C05487=1178.602,249.127,-64.757,-177.311,7.252,148.580
C05488=1178.597,249.375,-64.784,-177.309,7.254,148.579
C05489=1178.592,249.624,-64.811,-177.306,7.257,148.579
C05490=1178.588,249.872,-64.838,-177.303,7.259,148.579
C05491=1178.584,250.121,-64.865,-177.301,7.262,148.579
C05492=1178.580,250.370,-64.892,-177.299,7.264,148.579
C05493=1178.575,250.618,-64.919,-177.295,7.267,148.579
C05494=1178.571,250.866,-64.946,-177.293,7.270,148.579
C05495=1178.566,251.115,-64.973,-177.290,7.272,148.578
C05496=1178.562,251.363,-65.000,-177.288,7.275,148.578
C05497=1178.557,251.612,-65.027,-177.285,7.276,148.578
C05498=1178.553,251.860,-65.054,-177.282,7.279,148.578
C05499=1178.549,252.109,-65.081,-177.280,7.282,148.578
C05500=1178.545,252.358,-65.108,-177.277,7.285,148.578
C05501=1178.540,252.606,-65.135,-177.274,7.287,148.578
C05502=1178.536,252.854,-65.163,-177.272,7.289,148.577
C05503=1178.531,253.103,-65.190,-177.269,7.292,148.577
C05504=1178.526,253.351,-65.217,-177.267,7.295,148.577
C05505=1178.522,253.600,-65.244,-177.264,7.297,148.577
C05506=1178.518,253.849,-65.271,-177.261,7.300,148.577
C05507=1178.514,254.097,-65.298,-177.259,7.302,148.577
C05508=1178.509,254.345,-65.326,-177.256,7.305,148.577
C05509=1178.505,254.593,-65.353,-177.253,7.308,148.577
C05510=1178.500,254.842,-65.380,-177.251,7.310,148.576
C05511=1178.496,255.091,-65.407,-177.248,7.313,148.576
C05512=1178.492,255.339,-65.435,-177.245,7.316,148.576
C05513=1178.487,255.588,-65.462,-177.243,7.318,148.576
C05514=1178.482,255.836,-65.489,-177.240,7.321,148.576
C05515=1178.478,256.085,-65.517,-177.238,7.323,148.576
C05516=1178.474,256.333,-65.544,-177.235,7.326,148.576
C05517=1178.469,256.582,-65.571,-177.232,7.329,148.576
C05518=1178.464,256.830,-65.598,-177.230,7.331,148.575
C05519=1178.461,257.079,-65.627,-177.227,7.334,148.575
C05520=1178.456,257.327,-65.654,-177.224,7.337,148.575
C05521=1178.451,257.576,-65.681,-177.222,7.339,148.575
C05522=1178.447,257.824,-65.708,-177.219,7.342,148.575
C05523=1178.443,258.073,-65.736,-177.216,7.344,148.575
C05524=1178.438,258.321,-65.763,-177.214,7.347,148.575
C05525=1178.434,258.569,-65.791,-177.211,7.350,148.575
C05526=1178.429,258.818,-65.818,-177.209,7.352,148.575
C05527=1178.426,259.066,-65.846,-177.206,7.355,148.575
C05528=1178.421,259.315,-65.873,-177.204,7.358,148.575
C05529=1178.417,259.563,-65.901,-177.201,7.359,148.574
C05530=1178.413,259.812,-65.928,-177.198,7.362,148.574
C05531=1178.408,260.060,-65.956,-177.195,7.365,148.574
C05532=1178.404,260.308,-65.983,-177.193,7.368,148.574
C05533=1178.400,260.557,-66.011,-177.191,7.371,148.574
C05534=1178.394,260.805,-66.039,-177.188,7.373,148.574
C05535=1178.390,261.053,-66.067,-177.185,7.375,148.574
C05536=1178.386,261.303,-66.094,-177.182,7.378,148.574
C05537=1178.382,261.550,-66.122,-177.180,7.381,148.574
C05538=1178.377,261.799,-66.149,-177.177,7.383,148.573
C05539=1178.372,262.072,-66.180,-177.175,7.386,148.573
C05540=1178.367,262.345,-66.210,-177.172,7.389,148.573
C05541=1178.362,262.618,-66.241,-177.169,7.392,148.573
C05542=1178.358,262.891,-66.272,-177.165,7.396,148.573
C05543=1178.353,263.139,-66.299,-177.163,7.398,148.573
C05544=1178.349,263.387,-66.327,-177.161,7.401,148.573
C05545=1178.345,263.636,-66.354,-177.157,7.404,148.573
C05546=1178.341,263.884,-66.382,-177.155,7.406,148.573
C05547=1178.336,264.133,-66.411,-177.152,7.409,148.573
C05548=1178.332,264.381,-66.439,-177.150,7.412,148.573
C05549=1178.327,264.630,-66.466,-177.148,7.414,148.572
C05550=1178.323,264.878,-66.494,-177.145,7.417,148.572
C05551=1178.318,265.126,-66.522,-177.142,7.420,148.572
C05552=1178.315,265.375,-66.550,-177.140,7.422,148.572
C05553=1178.310,265.623,-66.577,-177.137,7.425,148.572
C05554=1178.306,265.871,-66.605,-177.134,7.428,148.572
C05555=1178.301,266.120,-66.634,-177.132,7.430,148.572
C05556=1178.297,266.368,-66.662,-177.129,7.433,148.572
C05557=1178.293,266.617,-66.690,-177.126,7.436,148.572
C05558=1178.288,266.865,-66.717,-177.124,7.439,148.572
C05559=1178.284,267.114,-66.746,-177.121,7.441,148.572
C05560=1178.279,267.362,-66.773,-177.119,7.444,148.572
C05561=1178.274,267.610,-66.802,-177.116,7.447,148.572
C05562=1178.271,267.859,-66.830,-177.114,7.449,148.571
C05563=1178.266,268.107,-66.858,-177.111,7.452,148.571
C05564=1178.262,268.355,-66.886,-177.108,7.455,148.571
C05565=1178.257,268.603,-66.914,-177.105,7.458,148.571
C05566=1178.253,268.853,-66.942,-177.103,7.460,148.571
C05567=1178.248,269.101,-66.970,-177.100,7.463,148.571
C05568=1178.245,269.349,-66.998,-177.097,7.466,148.571
C05569=1178.239,269.597,-67.026,-177.095,7.468,148.571
C05570=1178.236,269.846,-67.055,-177.093,7.471,148.571
C05571=1178.231,270.094,-67.083,-177.090,7.474,148.571
C05572=1178.227,270.343,-67.111,-177.087,7.477,148.571
C05573=1178.223,270.591,-67.139,-177.085,7.479,148.571
C05574=1178.218,270.840,-67.168,-177.082,7.482,148.571
C05575=1178.214,271.087,-67.195,-177.079,7.485,148.570
C05576=1178.209,271.336,-67.225,-177.077,7.487,148.570
C05577=1178.206,271.584,-67.253,-177.075,7.490,148.570
C05578=1178.201,271.832,-67.281,-177.072,7.493,148.570
C05579=1178.197,272.081,-67.309,-177.069,7.496,148.570
C05580=1178.192,272.329,-67.338,-177.066,7.498,148.570
C05581=1178.188,272.578,-67.366,-177.064,7.501,148.570
C05582=1178.183,272.826,-67.394,-177.061,7.504,148.570
C05583=1178.179,273.075,-67.423,-177.058,7.507,148.570
C05584=1178.174,273.322,-67.452,-177.056,7.509,148.570
C05585=1178.171,273.571,-67.480,-177.053,7.512,148.570
C05586=1178.166,273.820,-67.508,-177.051,7.515,148.570
C05587=1178.161,274.068,-67.537,-177.048,7.518,148.570
C05588=1178.157,274.316,-67.565,-177.046,7.520,148.570
C05589=1178.153,274.564,-67.594,-177.043,7.523,148.569
C05590=1178.149,274.813,-67.622,-177.040,7.526,148.569
C05591=1178.144,275.061,-67.651,-177.037,7.529,148.569
C05592=1178.140,275.309,-67.679,-177.035,7.531,148.569
C05593=1178.136,275.558,-67.708,-177.033,7.534,148.569
C05594=1178.131,275.806,-67.737,-177.030,7.537,148.569
C05595=1178.127,276.054,-67.765,-177.027,7.540,148.569
C05596=1178.123,276.303,-67.794,-177.025,7.542,148.569
C05597=1178.118,276.550,-67.822,-177.022,7.545,148.569
C05598=1178.114,276.799,-67.851,-177.019,7.548,148.569
C05599=1178.110,277.048,-67.880,-177.017,7.551,148.569
C05600=1178.105,277.295,-67.908,-177.015,7.553,148.569
C05601=1178.101,277.544,-67.937,-177.012,7.556,148.569
C05602=1178.097,277.793,-67.966,-177.009,7.559,148.569
C05603=1178.093,278.041,-67.994,-177.006,7.562,148.569
C05604=1178.088,278.289,-68.023,-177.004,7.565,148.569
C05605=1178.084,278.538,-68.052,-177.001,7.567,148.569
C05606=1178.080,278.786,-68.082,-176.999,7.570,148.569
C05607=1178.075,279.034,-68.109,-176.996,7.573,148.569
C05608=1178.071,279.283,-68.138,-176.993,7.576,148.569
C05609=1178.067,279.531,-68.167,-176.991,7.578,148.568
C05610=1178.062,279.779,-68.195,-176.988,7.581,148.568
C05611=1178.058,280.027,-68.225,-176.986,7.584,148.568
C05612=1178.054,280.275,-68.254,-176.983,7.587,148.568
C05613=1178.049,280.524,-68.283,-176.980,7.590,148.568
C05614=1178.045,280.772,-68.311,-176.978,7.592,148.568
C05615=1178.041,281.020,-68.340,-176.975,7.595,148.568
C05616=1178.037,281.269,-68.370,-176.973,7.598,148.568
C05617=1178.032,281.518,-68.398,-176.970,7.602,148.568
C05618=1178.027,281.765,-68.427,-176.968,7.604,148.568
C05619=1178.023,282.013,-68.457,-176.965,7.607,148.568
C05620=1178.019,282.262,-68.485,-176.963,7.610,148.568
C05621=1178.015,282.510,-68.514,-176.960,7.613,148.568
C05622=1178.010,282.758,-68.543,-176.957,7.616,148.568
C05623=1178.006,283.007,-68.572,-176.955,7.618,148.568
C05624=1178.002,283.255,-68.602,-176.952,7.621,148.568
C05625=1177.998,283.503,-68.631,-176.950,7.624,148.568
C05626=1177.993,283.751,-68.660,-176.947,7.627,148.568
C05627=1177.988,284.000,-68.689,-176.944,7.630,148.568
C05628=1177.985,284.248,-68.718,-176.942,7.632,148.568
C05629=1177.980,284.497,-68.747,-176.939,7.635,148.568
C05630=1177.976,284.745,-68.776,-176.936,7.638,148.568
C05631=1177.971,284.992,-68.805,-176.934,7.641,148.568
C05632=1177.967,285.241,-68.835,-176.931,7.644,148.568
C05633=1177.963,285.489,-68.864,-176.929,7.647,148.568
C05634=1177.959,285.738,-68.893,-176.927,7.649,148.568
C05635=1177.954,285.986,-68.922,-176.924,7.652,148.568
C05636=1177.950,286.234,-68.952,-176.921,7.655,148.568
C05637=1177.945,286.482,-68.981,-176.918,7.658,148.568
C05638=1177.941,286.730,-69.010,-176.916,7.661,148.568
C05639=1177.937,286.978,-69.040,-176.913,7.664,148.568
C05640=1177.933,287.227,-69.069,-176.911,7.667,148.568
C05641=1177.928,287.476,-69.098,-176.908,7.670,148.567
C05642=1177.924,287.724,-69.127,-176.905,7.673,148.567
C05643=1177.920,287.998,-69.160,-176.903,7.675,148.567
C05644=1177.915,288.273,-69.192,-176.900,7.679,148.568
C05645=1177.910,288.548,-69.226,-176.897,7.683,148.568
C05646=1177.905,288.822,-69.257,-176.894,7.686,148.568
C05647=1177.901,289.070,-69.287,-176.892,7.689,148.568
C05648=1177.897,289.319,-69.316,-176.889,7.692,148.568
C05649=1177.892,289.567,-69.346,-176.887,7.694,148.567
C05650=1177.888,289.815,-69.376,-176.884,7.697,148.567
C05651=1177.884,290.064,-69.405,-176.881,7.700,148.567
C05652=1177.880,290.312,-69.435,-176.878,7.703,148.567
C05653=1177.875,290.560,-69.464,-176.876,7.706,148.567
C05654=1177.871,290.809,-69.493,-176.873,7.709,148.567
C05655=1177.867,291.057,-69.523,-176.871,7.711,148.567
C05656=1177.863,291.304,-69.553,-176.869,7.714,148.567
C05657=1177.858,291.552,-69.582,-176.866,7.717,148.567
C05658=1177.853,291.801,-69.612,-176.863,7.720,148.567
C05659=1177.849,292.049,-69.642,-176.860,7.723,148.567
C05660=1177.845,292.297,-69.671,-176.858,7.726,148.567
C05661=1177.841,292.545,-69.701,-176.855,7.729,148.567
C05662=1177.837,292.794,-69.730,-176.853,7.732,148.567
C05663=1177.833,293.041,-69.760,-176.850,7.734,148.567
C05664=1177.828,293.290,-69.790,-176.848,7.737,148.567
C05665=1177.824,293.538,-69.820,-176.845,7.740,148.567
C05666=1177.820,293.786,-69.849,-176.842,7.743,148.567
C05667=1177.816,294.034,-69.879,-176.840,7.747,148.567
C05668=1177.811,294.283,-69.909,-176.837,7.750,148.567
C05669=1177.807,294.531,-69.939,-176.835,7.752,148.567
C05670=1177.802,294.779,-69.968,-176.832,7.755,148.567
C05671=1177.798,295.027,-69.998,-176.830,7.758,148.567
C05672=1177.794,295.275,-70.029,-176.827,7.761,148.567
C05673=1177.789,295.524,-70.058,-176.825,7.764,148.567
C05674=1177.785,295.771,-70.088,-176.822,7.767,148.567
C05675=1177.782,296.020,-70.118,-176.819,7.770,148.567
C05676=1177.777,296.269,-70.148,-176.816,7.773,148.567
C05677=1177.773,296.517,-70.178,-176.814,7.775,148.567
C05678=1177.769,296.765,-70.208,-176.812,7.779,148.567
C05679=1177.764,297.013,-70.238,-176.809,7.782,148.567
C05680=1177.760,297.261,-70.268,-176.807,7.785,148.567
C05681=1177.756,297.509,-70.297,-176.804,7.788,148.567
C05682=1177.751,297.757,-70.328,-176.801,7.791,148.567
C05683=1177.747,298.006,-70.358,-176.799,7.794,148.568
C05684=1177.743,298.253,-70.388,-176.796,7.797,148.568
C05685=1177.738,298.502,-70.418,-176.794,7.799,148.567
C05686=1177.734,298.749,-70.448,-176.791,7.802,148.567
C05687=1177.730,298.998,-70.478,-176.789,7.805,148.568
C05688=1177.726,299.246,-70.508,-176.786,7.808,148.568
C05689=1177.722,299.495,-70.538,-176.784,7.811,148.568
C05690=1177.718,299.743,-70.569,-176.781,7.814,148.568
C05691=1177.714,299.990,-70.599,-176.778,7.817,148.568
C05692=1177.709,300.239,-70.629,-176.776,7.821,148.568
C05693=1177.705,300.486,-70.659,-176.773,7.824,148.568
C05694=1177.700,300.735,-70.689,-176.771,7.826,148.568
C05695=1177.697,300.983,-70.720,-176.768,7.829,148.568
C05696=1177.692,301.231,-70.750,-176.766,7.832,148.568
C05697=1177.688,301.480,-70.780,-176.763,7.835,148.568
C05698=1177.684,301.727,-70.810,-176.760,7.838,148.568
C05699=1177.679,301.976,-70.840,-176.758,7.841,148.568
C05700=1177.675,302.223,-70.870,-176.755,7.844,148.568
C05701=1177.671,302.471,-70.901,-176.753,7.847,148.568
C05702=1177.667,302.720,-70.932,-176.750,7.850,148.568
C05703=1177.662,302.968,-70.962,-176.747,7.853,148.568
C05704=1177.658,303.216,-70.992,-176.746,7.856,148.568
C05705=1177.654,303.464,-71.023,-176.743,7.859,148.568
C05706=1177.649,303.712,-71.053,-176.740,7.862,148.568
C05707=1177.646,303.961,-71.083,-176.738,7.865,148.568
C05708=1177.641,304.209,-71.114,-176.735,7.868,148.568
C05709=1177.636,304.457,-71.145,-176.732,7.871,148.568
C05710=1177.633,304.704,-71.175,-176.730,7.874,148.568
C05711=1177.628,304.953,-71.205,-176.727,7.877,148.568
C05712=1177.624,305.201,-71.235,-176.725,7.880,148.568
C05713=1177.620,305.449,-71.266,-176.722,7.883,148.568
C05714=1177.615,305.697,-71.297,-176.720,7.887,148.568
C05715=1177.611,305.945,-71.327,-176.717,7.890,148.568
C05716=1177.607,306.194,-71.358,-176.715,7.892,148.568
C05717=1177.603,306.442,-71.389,-176.712,7.895,148.568
C05718=1177.599,306.689,-71.419,-176.710,7.898,148.569
C05719=1177.594,306.937,-71.450,-176.707,7.901,148.568
C05720=1177.590,307.186,-71.480,-176.704,7.904,148.568
C05721=1177.586,307.434,-71.511,-176.702,7.907,148.569
C05722=1177.581,307.682,-71.541,-176.699,7.910,148.569
C05723=1177.577,307.930,-71.572,-176.697,7.913,148.569
C05724=1177.573,308.178,-71.603,-176.694,7.917,148.569
C05725=1177.569,308.426,-71.633,-176.692,7.920,148.569
C05726=1177.564,308.674,-71.664,-176.689,7.923,148.569
C05727=1177.560,308.923,-71.695,-176.687,7.926,148.569
C05728=1177.557,309.170,-71.726,-176.684,7.929,148.569
C05729=1177.552,309.418,-71.757,-176.681,7.932,148.569
C05730=1177.548,309.667,-71.788,-176.679,7.934,148.569
C05731=1177.543,309.914,-71.819,-176.677,7.937,148.569
C05732=1177.540,310.162,-71.849,-176.674,7.940,148.569
C05733=1177.536,310.411,-71.880,-176.672,7.944,148.569
C05734=1177.531,310.659,-71.911,-176.669,7.947,148.569
C05735=1177.526,310.907,-71.942,-176.666,7.950,148.569
C05736=1177.522,311.155,-71.973,-176.664,7.953,148.569
C05737=1177.519,311.402,-72.004,-176.661,7.956,148.569
C05738=1177.514,311.650,-72.034,-176.659,7.959,148.569
C05739=1177.510,311.899,-72.066,-176.656,7.962,148.570
C05740=1177.505,312.147,-72.096,-176.654,7.965,148.570
C05741=1177.501,312.395,-72.127,-176.651,7.968,148.570
C05742=1177.497,312.643,-72.159,-176.649,7.971,148.570
C05743=1177.493,312.891,-72.190,-176.646,7.974,148.570
C05744=1177.489,313.139,-72.220,-176.644,7.978,148.570
C05745=1177.485,313.387,-72.251,-176.641,7.981,148.570
C05746=1177.480,313.635,-72.282,-176.639,7.984,148.570
C05747=1177.475,313.912,-72.317,-176.636,7.987,148.570
C05748=1177.471,314.189,-72.352,-176.633,7.990,148.570
C05749=1177.466,314.465,-72.387,-176.630,7.994,148.570
C05750=1177.462,314.742,-72.421,-176.628,7.997,148.570
C05751=1177.458,314.990,-72.453,-176.625,8.000,148.570
C05752=1177.453,315.238,-72.483,-176.623,8.003,148.570
C05753=1177.449,315.486,-72.515,-176.620,8.006,148.570
C05754=1177.445,315.734,-72.546,-176.617,8.009,148.570
C05755=1177.440,315.982,-72.577,-176.615,8.013,148.571
C05756=1177.437,316.230,-72.609,-176.612,8.016,148.571
C05757=1177.432,316.478,-72.639,-176.610,8.019,148.571
C05758=1177.428,316.726,-72.671,-176.607,8.022,148.571
C05759=1177.424,316.974,-72.702,-176.605,8.025,148.571
C05760=1177.420,317.222,-72.734,-176.602,8.028,148.571
C05761=1177.415,317.470,-72.765,-176.599,8.031,148.571
C05762=1177.412,317.718,-72.796,-176.597,8.035,148.571
C05763=1177.407,317.966,-72.827,-176.594,8.038,148.571
C05764=1177.403,318.214,-72.859,-176.592,8.041,148.571
C05765=1177.399,318.462,-72.890,-176.589,8.044,148.571
C05766=1177.395,318.710,-72.922,-176.587,8.047,148.572
C05767=1177.391,318.958,-72.953,-176.584,8.050,148.572
C05768=1177.387,319.206,-72.984,-176.582,8.053,148.572
C05769=1177.382,319.454,-73.016,-176.579,8.056,148.572
C05770=1177.378,319.703,-73.047,-176.577,8.060,148.572
C05771=1177.373,319.950,-73.079,-176.574,8.063,148.572
C05772=1177.370,320.198,-73.111,-176.572,8.066,148.572
C05773=1177.365,320.446,-73.142,-176.569,8.069,148.572
C05774=1177.361,320.694,-73.173,-176.567,8.072,148.572
C05775=1177.358,320.942,-73.205,-176.564,8.075,148.572
C05776=1177.353,321.190,-73.236,-176.562,8.079,148.573
C05777=1177.349,321.438,-73.268,-176.559,8.082,148.573
C05778=1177.344,321.686,-73.300,-176.557,8.085,148.573
C05779=1177.340,321.934,-73.331,-176.555,8.088,148.573
C05780=1177.336,322.182,-73.363,-176.552,8.091,148.573
C05781=1177.332,322.430,-73.394,-176.550,8.094,148.573
C05782=1177.328,322.678,-73.426,-176.547,8.098,148.573
C05783=1177.324,322.925,-73.458,-176.545,8.101,148.573
C05784=1177.319,323.174,-73.489,-176.542,8.104,148.573
C05785=1177.315,323.422,-73.521,-176.540,8.107,148.573
C05786=1177.311,323.670,-73.553,-176.537,8.110,148.574
C05787=1177.308,323.918,-73.585,-176.535,8.113,148.574
C05788=1177.303,324.165,-73.617,-176.532,8.116,148.574
C05789=1177.299,324.413,-73.649,-176.530,8.119,148.574
C05790=1177.295,324.662,-73.680,-176.527,8.123,148.574
C05791=1177.291,324.909,-73.711,-176.525,8.126,148.574
C05792=1177.286,325.158,-73.744,-176.522,8.129,148.574
C05793=1177.282,325.406,-73.775,-176.520,8.132,148.574
C05794=1177.278,325.653,-73.807,-176.517,8.135,148.574
C05795=1177.274,325.901,-73.839,-176.515,8.139,148.575
C05796=1177.270,326.149,-73.871,-176.512,8.142,148.574
C05797=1177.266,326.397,-73.903,-176.510,8.145,148.575
C05798=1177.261,326.645,-73.935,-176.507,8.148,148.575
C05799=1177.258,326.893,-73.967,-176.505,8.151,148.575
C05800=1177.253,327.140,-73.998,-176.503,8.155,148.575
C05801=1177.249,327.389,-74.031,-176.500,8.158,148.575
C05802=1177.245,327.637,-74.063,-176.498,8.161,148.575
C05803=1177.241,327.884,-74.094,-176.495,8.164,148.575
C05804=1177.236,328.133,-74.127,-176.493,8.167,148.576
C05805=1177.233,328.381,-74.158,-176.491,8.171,148.576
C05806=1177.228,328.628,-74.190,-176.488,8.174,148.576
C05807=1177.224,328.876,-74.222,-176.486,8.177,148.576
C05808=1177.221,329.124,-74.255,-176.483,8.180,148.576
C05809=1177.216,329.372,-74.287,-176.481,8.183,148.576
C05810=1177.212,329.619,-74.319,-176.478,8.186,148.576
C05811=1177.207,329.868,-74.351,-176.476,8.189,148.576
C05812=1177.204,330.116,-74.383,-176.473,8.193,148.577
C05813=1177.199,330.364,-74.416,-176.471,8.196,148.577
C05814=1177.195,330.611,-74.448,-176.468,8.199,148.577
C05815=1177.191,330.859,-74.480,-176.466,8.202,148.577
C05816=1177.187,331.107,-74.512,-176.464,8.206,148.577
C05817=1177.183,331.356,-74.545,-176.461,8.209,148.577
C05818=1177.179,331.602,-74.577,-176.459,8.212,148.577
C05819=1177.174,331.851,-74.609,-176.456,8.215,148.578
C05820=1177.170,332.099,-74.641,-176.454,8.218,148.578
C05821=1177.166,332.347,-74.673,-176.451,8.222,148.578
C05822=1177.162,332.594,-74.706,-176.449,8.225,148.578
C05823=1177.158,332.842,-74.738,-176.446,8.229,148.578
C05824=1177.154,333.090,-74.770,-176.444,8.232,148.578
C05825=1177.150,333.338,-74.803,-176.441,8.235,148.578
C05826=1177.146,333.586,-74.835,-176.439,8.238,148.578
C05827=1177.142,333.834,-74.867,-176.436,8.242,148.579
C05828=1177.137,334.081,-74.900,-176.434,8.245,148.579
C05829=1177.133,334.329,-74.932,-176.432,8.248,148.579
C05830=1177.129,334.577,-74.965,-176.429,8.251,148.579
C05831=1177.125,334.825,-74.997,-176.427,8.255,148.579
C05832=1177.121,335.073,-75.029,-176.425,8.258,148.579
C05833=1177.117,335.321,-75.063,-176.422,8.261,148.580
C05834=1177.112,335.568,-75.094,-176.420,8.264,148.580
C05835=1177.108,335.816,-75.127,-176.417,8.267,148.580
C05836=1177.104,336.065,-75.160,-176.415,8.271,148.580
C05837=1177.100,336.312,-75.192,-176.413,8.274,148.580
C05838=1177.096,336.560,-75.225,-176.410,8.277,148.580
C05839=1177.092,336.808,-75.258,-176.408,8.280,148.581
C05840=1177.088,337.056,-75.290,-176.406,8.284,148.581
C05841=1177.084,337.304,-75.323,-176.403,8.287,148.581
C05842=1177.079,337.551,-75.356,-176.400,8.291,148.581
C05843=1177.076,337.799,-75.387,-176.398,8.294,148.581
C05844=1177.071,338.047,-75.421,-176.395,8.297,148.581
C05845=1177.067,338.295,-75.453,-176.393,8.301,148.582
C05846=1177.063,338.543,-75.486,-176.391,8.304,148.582
C05847=1177.059,338.790,-75.519,-176.388,8.307,148.582
C05848=1177.055,339.038,-75.551,-176.386,8.310,148.582
C05849=1177.051,339.286,-75.584,-176.384,8.314,148.582
C05850=1177.047,339.534,-75.618,-176.381,8.317,148.582
C05851=1177.042,339.812,-75.654,-176.379,8.321,148.583
C05852=1177.037,340.093,-75.691,-176.376,8.324,148.583
C05853=1177.033,340.371,-75.727,-176.373,8.328,148.583
C05854=1177.028,340.651,-75.765,-176.371,8.332,148.583
C05855=1177.024,340.899,-75.798,-176.368,8.336,148.583
C05856=1177.021,341.146,-75.831,-176.366,8.339,148.584
C05857=1177.016,341.394,-75.863,-176.363,8.342,148.584
C05858=1177.012,341.641,-75.896,-176.361,8.346,148.584
C05859=1177.007,341.889,-75.929,-176.359,8.349,148.584
C05860=1177.003,342.137,-75.962,-176.357,8.352,148.585
C05861=1176.999,342.385,-75.995,-176.354,8.355,148.585
C05862=1176.995,342.633,-76.028,-176.352,8.358,148.585
C05863=1176.991,342.881,-76.061,-176.349,8.362,148.585
C05864=1176.987,343.128,-76.094,-176.347,8.365,148.585
C05865=1176.983,343.376,-76.127,-176.345,8.368,148.585
C05866=1176.979,343.623,-76.160,-176.342,8.373,148.586
C05867=1176.975,343.871,-76.193,-176.340,8.376,148.586
C05868=1176.971,344.119,-76.226,-176.337,8.379,148.586
C05869=1176.966,344.367,-76.259,-176.335,8.382,148.586
C05870=1176.962,344.614,-76.293,-176.333,8.386,148.587
C05871=1176.959,344.863,-76.326,-176.331,8.389,148.587
C05872=1176.955,345.111,-76.359,-176.328,8.392,148.587
C05873=1176.950,345.358,-76.392,-176.326,8.396,148.587
C05874=1176.946,345.606,-76.426,-176.324,8.399,148.587
C05875=1176.942,345.854,-76.459,-176.321,8.402,148.588
C05876=1176.938,346.101,-76.492,-176.319,8.406,148.588
C05877=1176.934,346.349,-76.525,-176.316,8.410,148.588
C05878=1176.930,346.597,-76.558,-176.314,8.413,148.588
C05879=1176.926,346.845,-76.591,-176.312,8.416,148.589
C05880=1176.922,347.092,-76.624,-176.310,8.420,148.589
C05881=1176.917,347.340,-76.658,-176.307,8.423,148.589
C05882=1176.913,347.588,-76.691,-176.305,8.426,148.589
C05883=1176.909,347.836,-76.724,-176.303,8.430,148.589
C05884=1176.905,348.083,-76.757,-176.300,8.433,148.590
C05885=1176.902,348.331,-76.791,-176.298,8.437,148.590
C05886=1176.898,348.579,-76.824,-176.295,8.440,148.590
C05887=1176.893,348.827,-76.858,-176.293,8.444,148.590
C05888=1176.889,349.075,-76.891,-176.291,8.447,148.591
C05889=1176.884,349.322,-76.925,-176.289,8.451,148.591
C05890=1176.881,349.569,-76.958,-176.287,8.454,148.591
C05891=1176.876,349.817,-76.992,-176.284,8.457,148.591
C05892=1176.872,350.065,-77.025,-176.282,8.461,148.592
C05893=1176.869,350.313,-77.058,-176.279,8.465,148.592
C05894=1176.865,350.560,-77.092,-176.277,8.468,148.592
C05895=1176.860,350.809,-77.126,-176.275,8.471,148.592
C05896=1176.856,351.056,-77.159,-176.272,8.475,148.593
C05897=1176.852,351.304,-77.192,-176.271,8.478,148.593
C05898=1176.848,351.551,-77.226,-176.268,8.481,148.593
C05899=1176.844,351.800,-77.260,-176.266,8.485,148.593
C05900=1176.840,352.047,-77.293,-176.264,8.488,148.594
C05901=1176.836,352.295,-77.327,-176.261,8.492,148.594
C05902=1176.832,352.542,-77.360,-176.259,8.496,148.594
C05903=1176.828,352.789,-77.394,-176.257,8.499,148.595
C05904=1176.824,353.038,-77.428,-176.255,8.502,148.595
C05905=1176.819,353.286,-77.461,-176.252,8.506,148.595
C05906=1176.816,353.533,-77.495,-176.250,8.509,148.595
C05907=1176.811,353.781,-77.529,-176.248,8.513,148.596
C05908=1176.808,354.028,-77.562,-176.245,8.517,148.596
C05909=1176.803,354.277,-77.596,-176.243,8.520,148.596
C05910=1176.799,354.524,-77.630,-176.241,8.523,148.596
C05911=1176.795,354.771,-77.664,-176.239,8.527,148.597
C05912=1176.791,355.019,-77.697,-176.237,8.530,148.597
C05913=1176.787,355.267,-77.732,-176.235,8.534,148.597
C05914=1176.783,355.514,-77.765,-176.232,8.538,148.597
C05915=1176.779,355.762,-77.799,-176.230,8.541,148.598
C05916=1176.775,356.010,-77.833,-176.228,8.545,148.598
C05917=1176.771,356.257,-77.867,-176.225,8.548,148.598
C05918=1176.767,356.505,-77.900,-176.223,8.552,148.599
C05919=1176.763,356.753,-77.935,-176.221,8.555,148.599
C05920=1176.759,357.001,-77.968,-176.218,8.559,148.599
C05921=1176.755,357.248,-78.002,-176.217,8.563,148.600
C05922=1176.751,357.496,-78.037,-176.214,8.566,148.600
C05923=1176.747,357.744,-78.070,-176.212,8.569,148.600
C05924=1176.743,357.991,-78.105,-176.210,8.573,148.601
C05925=1176.739,358.238,-78.139,-176.208,8.576,148.601
C05926=1176.735,358.486,-78.172,-176.206,8.581,148.601
C05927=1176.731,358.734,-78.207,-176.203,8.584,148.601
C05928=1176.727,358.981,-78.240,-176.201,8.588,148.602
C05929=1176.722,359.229,-78.275,-176.199,8.591,148.602
C05930=1176.719,359.477,-78.308,-176.197,8.594,148.602
C05931=1176.715,359.724,-78.342,-176.195,8.598,148.603
C05932=1176.711,359.973,-78.377,-176.193,8.601,148.603
C05933=1176.707,360.220,-78.411,-176.190,8.606,148.603
C05934=1176.702,360.468,-78.445,-176.189,8.609,148.604
C05935=1176.699,360.715,-78.479,-176.186,8.613,148.604
C05936=1176.694,360.963,-78.513,-176.184,8.616,148.605
C05937=1176.691,361.210,-78.547,-176.182,8.619,148.605
C05938=1176.687,361.458,-78.582,-176.180,8.623,148.605
C05939=1176.683,361.705,-78.616,-176.178,8.626,148.605
C05940=1176.679,361.953,-78.651,-176.176,8.630,148.606
C05941=1176.675,362.201,-78.684,-176.174,8.634,148.606
C05942=1176.670,362.448,-78.718,-176.172,8.638,148.607
C05943=1176.667,362.696,-78.753,-176.170,8.641,148.607
C05944=1176.662,362.944,-78.787,-176.168,8.645,148.607
C05945=1176.659,363.192,-78.821,-176.166,8.648,148.608
C05946=1176.655,363.439,-78.856,-176.164,8.652,148.608
C05947=1176.650,363.686,-78.890,-176.162,8.655,148.608
C05948=1176.647,363.934,-78.925,-176.160,8.659,148.609
C05949=1176.642,364.182,-78.959,-176.158,8.662,148.609
C05950=1176.639,364.429,-78.993,-176.156,8.666,148.610
C05951=1176.634,364.677,-79.028,-176.154,8.670,148.610
C05952=1176.631,364.925,-79.062,-176.152,8.673,148.610
C05953=1176.627,365.172,-79.096,-176.150,8.678,148.611
C05954=1176.623,365.420,-79.131,-176.148,8.681,148.611
C05955=1176.618,365.702,-79.170,-176.146,8.685,148.612
C05956=1176.614,365.983,-79.210,-176.144,8.689,148.612
C05957=1176.609,366.265,-79.249,-176.142,8.693,148.613
C05958=1176.605,366.547,-79.288,-176.140,8.697,148.613
C05959=1176.601,366.794,-79.323,-176.138,8.701,148.614
C05960=1176.597,367.042,-79.358,-176.136,8.705,148.614
C05961=1176.592,367.290,-79.392,-176.134,8.708,148.614
C05962=1176.588,367.537,-79.426,-176.132,8.712,148.615
C05963=1176.585,367.784,-79.461,-176.131,8.715,148.615
C05964=1176.580,368.032,-79.496,-176.129,8.719,148.616
C05965=1176.577,368.280,-79.530,-176.127,8.723,148.616
C05966=1176.572,368.527,-79.565,-176.125,8.727,148.617
C05967=1176.568,368.775,-79.599,-176.124,8.730,148.617
C05968=1176.565,369.023,-79.635,-176.122,8.734,148.618
C05969=1176.561,369.270,-79.669,-176.121,8.737,148.618
C05970=1176.557,369.518,-79.704,-176.119,8.740,148.618
C05971=1176.552,369.765,-79.738,-176.117,8.744,148.619
C05972=1176.549,370.013,-79.774,-176.115,8.748,148.620
C05973=1176.545,370.260,-79.808,-176.114,8.751,148.620
C05974=1176.541,370.508,-79.842,-176.112,8.755,148.620
C05975=1176.536,370.755,-79.878,-176.110,8.759,148.621
C05976=1176.533,371.003,-79.912,-176.109,8.763,148.621
C05977=1176.528,371.250,-79.947,-176.107,8.765,148.622
C05978=1176.525,371.498,-79.982,-176.106,8.769,148.622
C05979=1176.520,371.745,-80.016,-176.104,8.773,148.623
C05980=1176.516,371.993,-80.051,-176.103,8.777,148.624
C05981=1176.513,372.241,-80.087,-176.101,8.780,148.624
C05982=1176.508,372.488,-80.121,-176.100,8.783,148.625
C05983=1176.505,372.736,-80.157,-176.098,8.787,148.625
C05984=1176.501,372.983,-80.191,-176.097,8.791,148.626
C05985=1176.497,373.231,-80.225,-176.095,8.795,148.626
C05986=1176.493,373.478,-80.261,-176.094,8.798,148.627
C05987=1176.489,373.726,-80.295,-176.092,8.801,148.627
C05988=1176.485,373.973,-80.331,-176.091,8.805,148.628
C05989=1176.480,374.221,-80.365,-176.089,8.809,148.628
C05990=1176.477,374.468,-80.401,-176.088,8.812,148.629
C05991=1176.473,374.716,-80.436,-176.087,8.816,148.629
C05992=1176.469,374.963,-80.470,-176.085,8.819,148.630
C05993=1176.465,375.211,-80.505,-176.084,8.823,148.630
C05994=1176.461,375.458,-80.540,-176.083,8.826,148.631
C05995=1176.457,375.706,-80.575,-176.082,8.830,148.632
C05996=1176.453,375.953,-80.611,-176.080,8.833,148.632
C05997=1176.449,376.201,-80.645,-176.079,8.837,148.633
C05998=1176.445,376.448,-80.681,-176.078,8.840,148.633
C05999=1176.441,376.696,-80.716,-176.076,8.844,148.634
C06000=1176.437,376.943,-80.751,-176.076,8.847,148.634
C06001=1176.433,377.191,-80.786,-176.074,8.851,148.635
C06002=1176.429,377.439,-80.821,-176.073,8.854,148.635
C06003=1176.425,377.686,-80.856,-176.072,8.858,148.636
C06004=1176.421,377.933,-80.892,-176.071,8.861,148.637
C06005=1176.417,378.181,-80.927,-176.069,8.865,148.637
C06006=1176.413,378.428,-80.962,-176.069,8.868,148.638
C06007=1176.409,378.675,-80.998,-176.067,8.872,148.638
C06008=1176.405,378.924,-81.032,-176.066,8.875,148.639
C06009=1176.401,379.170,-81.068,-176.065,8.878,148.640
C06010=1176.398,379.418,-81.103,-176.064,8.882,148.640
C06011=1176.394,379.666,-81.138,-176.063,8.885,148.641
C06012=1176.389,379.913,-81.173,-176.062,8.888,148.641
C06013=1176.386,380.160,-81.209,-176.061,8.892,148.642
C06014=1176.382,380.408,-81.243,-176.060,8.895,148.643
C06015=1176.377,380.655,-81.279,-176.059,8.898,148.643
C06016=1176.374,380.903,-81.314,-176.058,8.902,148.644
C06017=1176.370,381.150,-81.350,-176.058,8.906,148.645
C06018=1176.366,381.398,-81.385,-176.057,8.909,148.645
C06019=1176.362,381.645,-81.420,-176.056,8.912,148.646
C06020=1176.358,381.893,-81.455,-176.055,8.916,148.646
C06021=1176.354,382.140,-81.491,-176.054,8.919,148.647
C06022=1176.349,382.387,-81.527,-176.053,8.922,148.648
C06023=1176.346,382.635,-81.561,-176.052,8.925,148.648
C06024=1176.342,382.883,-81.597,-176.052,8.928,148.649
C06025=1176.338,383.130,-81.633,-176.051,8.931,148.650
C06026=1176.334,383.377,-81.668,-176.050,8.935,148.650
C06027=1176.330,383.625,-81.703,-176.050,8.938,148.651
C06028=1176.327,383.872,-81.739,-176.048,8.942,148.651
C06029=1176.323,384.120,-81.774,-176.048,8.945,148.652
C06030=1176.318,384.367,-81.809,-176.047,8.948,148.653
C06031=1176.314,384.615,-81.845,-176.047,8.952,148.654
C06032=1176.310,384.862,-81.881,-176.046,8.955,148.654
C06033=1176.307,385.110,-81.916,-176.045,8.957,148.655
C06034=1176.302,385.357,-81.951,-176.045,8.960,148.656
C06035=1176.299,385.604,-81.987,-176.044,8.964,148.656
C06036=1176.295,385.852,-82.022,-176.044,8.967,148.657
C06037=1176.291,386.099,-82.058,-176.043,8.970,148.657
C06038=1176.286,386.347,-82.093,-176.043,8.973,148.658
C06039=1176.282,386.594,-82.129,-176.042,8.976,148.659
C06040=1176.279,386.842,-82.164,-176.041,8.980,148.660
C06041=1176.275,387.089,-82.200,-176.041,8.982,148.660
C06042=1176.271,387.336,-82.235,-176.041,8.986,148.661
C06043=1176.266,387.584,-82.271,-176.040,8.989,148.661
C06044=1176.263,387.832,-82.307,-176.039,8.992,148.662
C06045=1176.259,388.079,-82.342,-176.040,8.995,148.663
C06046=1176.255,388.327,-82.378,-176.039,8.998,148.664
C06047=1176.251,388.573,-82.413,-176.038,9.001,148.664
C06048=1176.247,388.821,-82.449,-176.038,9.003,148.665
C06049=1176.243,389.069,-82.484,-176.038,9.007,148.666
C06050=1176.239,389.316,-82.520,-176.038,9.009,148.666
C06051=1176.236,389.564,-82.556,-176.037,9.012,148.667
C06052=1176.232,389.810,-82.591,-176.037,9.015,148.668
C06053=1176.227,390.058,-82.627,-176.037,9.018,148.668
C06054=1176.223,390.306,-82.662,-176.037,9.021,148.669
C06055=1176.220,390.553,-82.698,-176.036,9.024,148.670
C06056=1176.216,390.801,-82.734,-176.036,9.027,148.670
C06057=1176.212,391.048,-82.769,-176.035,9.030,148.671
C06058=1176.207,391.295,-82.805,-176.036,9.032,148.672
C06059=1176.204,391.579,-82.846,-176.035,9.036,148.672
C06060=1176.199,391.864,-82.887,-176.035,9.039,148.673
C06061=1176.195,392.149,-82.928,-176.035,9.043,148.674
C06062=1176.190,392.433,-82.969,-176.035,9.045,148.675
C06063=1176.186,392.680,-83.004,-176.034,9.048,148.676
C06064=1176.182,392.927,-83.041,-176.034,9.051,148.676
C06065=1176.178,393.175,-83.077,-176.035,9.054,148.677
C06066=1176.174,393.423,-83.112,-176.035,9.056,148.678
C06067=1176.171,393.670,-83.148,-176.034,9.059,148.678
C06068=1176.166,393.917,-83.184,-176.034,9.062,148.679
C06069=1176.162,394.165,-83.219,-176.034,9.064,148.680
C06070=1176.158,394.412,-83.255,-176.034,9.067,148.680
C06071=1176.155,394.660,-83.290,-176.033,9.070,148.681
C06072=1176.151,394.907,-83.327,-176.034,9.073,148.682
C06073=1176.147,395.154,-83.363,-176.034,9.075,148.682
C06074=1176.143,395.402,-83.398,-176.034,9.078,148.683
C06075=1176.138,395.649,-83.434,-176.034,9.080,148.684
C06076=1176.135,395.896,-83.470,-176.034,9.083,148.684
C06077=1176.131,396.144,-83.505,-176.034,9.085,148.685
C06078=1176.127,396.392,-83.541,-176.034,9.088,148.686
C06079=1176.123,396.639,-83.578,-176.033,9.091,148.686
C06080=1176.120,396.886,-83.613,-176.034,9.093,148.687
C06081=1176.115,397.133,-83.649,-176.034,9.096,148.688
C06082=1176.111,397.381,-83.684,-176.034,9.098,148.689
C06083=1176.107,397.628,-83.720,-176.034,9.101,148.689
C06084=1176.103,397.875,-83.757,-176.034,9.103,148.690
C06085=1176.100,398.123,-83.792,-176.034,9.106,148.690
C06086=1176.096,398.370,-83.828,-176.034,9.108,148.691
C06087=1176.091,398.618,-83.864,-176.034,9.111,148.692
C06088=1176.087,398.865,-83.899,-176.035,9.112,148.692
C06089=1176.084,399.112,-83.936,-176.035,9.115,148.693
C06090=1176.079,399.360,-83.972,-176.035,9.118,148.694
C06091=1176.076,399.607,-84.007,-176.035,9.120,148.694
C06092=1176.072,399.855,-84.043,-176.035,9.122,148.695
C06093=1176.068,400.103,-84.079,-176.035,9.125,148.696
C06094=1176.064,400.349,-84.115,-176.035,9.127,148.696
C06095=1176.061,400.597,-84.151,-176.035,9.130,148.697
C06096=1176.056,400.844,-84.186,-176.035,9.132,148.698
C06097=1176.052,401.092,-84.222,-176.036,9.134,148.698
C06098=1176.049,401.338,-84.258,-176.035,9.136,148.699
C06099=1176.044,401.586,-84.294,-176.036,9.139,148.700
C06100=1176.041,401.834,-84.330,-176.036,9.141,148.700
C06101=1176.036,402.082,-84.366,-176.035,9.144,148.701
C06102=1176.033,402.328,-84.402,-176.036,9.145,148.702
C06103=1176.029,402.576,-84.438,-176.036,9.148,148.702
C06104=1176.025,402.824,-84.474,-176.036,9.150,148.703
C06105=1176.021,403.071,-84.509,-176.036,9.153,148.703
C06106=1176.017,403.317,-84.546,-176.037,9.155,148.704
C06107=1176.013,403.565,-84.582,-176.037,9.157,148.705
C06108=1176.009,403.813,-84.617,-176.037,9.159,148.705
C06109=1176.005,404.060,-84.654,-176.037,9.161,148.706
C06110=1176.001,404.307,-84.690,-176.037,9.163,148.707
C06111=1175.998,404.555,-84.725,-176.037,9.166,148.707
C06112=1175.993,404.803,-84.761,-176.038,9.167,148.708
C06113=1175.990,405.050,-84.798,-176.038,9.170,148.708
C06114=1175.986,405.297,-84.834,-176.038,9.172,148.709
C06115=1175.982,405.545,-84.869,-176.038,9.174,148.710
C06116=1175.978,405.791,-84.905,-176.039,9.177,148.710
C06117=1175.974,406.039,-84.941,-176.038,9.179,148.711
C06118=1175.970,406.286,-84.977,-176.039,9.181,148.711
C06119=1175.966,406.534,-85.014,-176.039,9.183,148.712
C06120=1175.962,406.781,-85.049,-176.039,9.185,148.713
C06121=1175.958,407.029,-85.085,-176.039,9.187,148.713
C06122=1175.954,407.276,-85.122,-176.039,9.189,148.714
C06123=1175.951,407.523,-85.157,-176.040,9.191,148.714
C06124=1175.946,407.771,-85.193,-176.040,9.193,148.715
C06125=1175.943,408.018,-85.230,-176.040,9.195,148.716
C06126=1175.939,408.266,-85.266,-176.040,9.197,148.716
C06127=1175.934,408.513,-85.301,-176.040,9.199,148.717
C06128=1175.931,408.759,-85.337,-176.041,9.201,148.717
C06129=1175.926,409.007,-85.373,-176.041,9.203,148.718
C06130=1175.923,409.255,-85.409,-176.041,9.205,148.719
C06131=1175.919,409.502,-85.446,-176.041,9.207,148.719
C06132=1175.915,409.750,-85.481,-176.042,9.209,148.720
C06133=1175.911,409.997,-85.518,-176.042,9.211,148.720
C06134=1175.907,410.244,-85.554,-176.042,9.213,148.721
C06135=1175.904,410.492,-85.589,-176.042,9.215,148.721
C06136=1175.900,410.739,-85.626,-176.042,9.217,148.722
C06137=1175.896,410.986,-85.662,-176.043,9.219,148.723
C06138=1175.891,411.234,-85.698,-176.042,9.221,148.723
C06139=1175.888,411.481,-85.734,-176.043,9.223,148.724
C06140=1175.884,411.729,-85.770,-176.043,9.225,148.724
C06141=1175.880,411.976,-85.806,-176.043,9.227,148.725
C06142=1175.875,412.223,-85.842,-176.043,9.229,148.725
C06143=1175.872,412.470,-85.878,-176.044,9.231,148.726
C06144=1175.868,412.718,-85.915,-176.044,9.232,148.726
C06145=1175.864,412.965,-85.950,-176.044,9.235,148.727
C06146=1175.861,413.212,-85.986,-176.044,9.236,148.727
C06147=1175.856,413.460,-86.023,-176.044,9.238,148.728
C06148=1175.853,413.707,-86.058,-176.045,9.240,148.729
C06149=1175.848,413.954,-86.095,-176.045,9.242,148.729
C06150=1175.845,414.202,-86.131,-176.045,9.244,148.730
C06151=1175.841,414.449,-86.167,-176.046,9.246,148.730
C06152=1175.837,414.697,-86.203,-176.045,9.248,148.731
C06153=1175.833,414.944,-86.240,-176.046,9.249,148.731
C06154=1175.829,415.191,-86.275,-176.045,9.251,148.732
C06155=1175.825,415.437,-86.311,-176.046,9.253,148.732
C06156=1175.821,415.682,-86.348,-176.046,9.255,148.733
C06157=1175.819,415.929,-86.383,-176.046,9.257,148.733
C06158=1175.818,416.174,-86.418,-176.046,9.258,148.734
C06159=1175.817,416.420,-86.454,-176.047,9.260,148.734
C06160=1175.818,416.665,-86.490,-176.046,9.262,148.735
C06161=1175.820,416.910,-86.525,-176.047,9.263,148.735
C06162=1175.823,417.155,-86.560,-176.047,9.265,148.736
C06163=1175.402,417.157,-86.604,-176.050,9.276,148.740
C06164=1175.399,416.910,-86.569,-176.050,9.274,148.739
C06165=1175.397,416.663,-86.532,-176.050,9.273,148.739
C06166=1175.396,416.416,-86.498,-176.050,9.271,148.738
C06167=1175.397,416.169,-86.461,-176.050,9.269,148.738
C06168=1175.398,415.922,-86.426,-176.049,9.268,148.737
C06169=1175.401,415.675,-86.389,-176.049,9.265,148.736
C06170=1175.404,415.427,-86.353,-176.049,9.264,148.736
C06171=1175.408,415.180,-86.317,-176.049,9.262,148.736
C06172=1175.412,414.933,-86.281,-176.049,9.260,148.735
C06173=1175.415,414.686,-86.245,-176.048,9.258,148.734
C06174=1175.420,414.438,-86.209,-176.048,9.256,148.734
C06175=1175.424,414.190,-86.173,-176.048,9.255,148.733
C06176=1175.428,413.943,-86.136,-176.047,9.253,148.733
C06177=1175.431,413.696,-86.101,-176.048,9.251,148.732
C06178=1175.435,413.449,-86.064,-176.047,9.249,148.732
C06179=1175.439,413.201,-86.028,-176.047,9.247,148.731
C06180=1175.442,412.954,-85.992,-176.047,9.245,148.731
C06181=1175.447,412.706,-85.956,-176.047,9.244,148.730
C06182=1175.450,412.459,-85.920,-176.047,9.241,148.729
C06183=1175.455,412.212,-85.883,-176.046,9.240,148.729
C06184=1175.458,411.964,-85.848,-176.047,9.238,148.728
C06185=1175.463,411.718,-85.811,-176.046,9.236,148.728
C06186=1175.467,411.470,-85.776,-176.046,9.234,148.727
C06187=1175.471,411.222,-85.740,-176.045,9.232,148.727
C06188=1175.474,410.976,-85.703,-176.046,9.230,148.726
C06189=1175.479,410.728,-85.667,-176.045,9.228,148.726
C06190=1175.482,410.481,-85.631,-176.045,9.226,148.725
C06191=1175.487,410.233,-85.595,-176.045,9.224,148.725
C06192=1175.490,409.985,-85.559,-176.044,9.222,148.724
C06193=1175.494,409.739,-85.523,-176.044,9.220,148.723
C06194=1175.498,409.491,-85.487,-176.044,9.218,148.723
C06195=1175.502,409.243,-85.451,-176.044,9.216,148.722
C06196=1175.506,408.996,-85.415,-176.044,9.215,148.722
C06197=1175.509,408.749,-85.379,-176.044,9.212,148.721
C06198=1175.513,408.501,-85.342,-176.043,9.211,148.721
C06199=1175.517,408.254,-85.307,-176.043,9.208,148.720
C06200=1175.521,408.007,-85.271,-176.043,9.206,148.719
C06201=1175.525,407.760,-85.235,-176.043,9.204,148.719
C06202=1175.529,407.512,-85.199,-176.043,9.202,148.718
C06203=1175.534,407.265,-85.163,-176.042,9.200,148.717
C06204=1175.537,407.018,-85.127,-176.042,9.198,148.717
C06205=1175.541,406.770,-85.090,-176.042,9.196,148.716
C06206=1175.545,406.522,-85.055,-176.042,9.194,148.716
C06207=1175.548,406.276,-85.019,-176.041,9.192,148.715
C06208=1175.553,406.028,-84.982,-176.041,9.190,148.714
C06209=1175.556,405.780,-84.947,-176.041,9.187,148.714
C06210=1175.560,405.533,-84.910,-176.041,9.186,148.713
C06211=1175.564,405.286,-84.875,-176.041,9.183,148.713
C06212=1175.568,405.039,-84.839,-176.041,9.181,148.712
C06213=1175.572,404.792,-84.802,-176.040,9.179,148.711
C06214=1175.576,404.544,-84.767,-176.040,9.177,148.711
C06215=1175.581,404.296,-84.731,-176.040,9.175,148.710
C06216=1175.584,404.049,-84.695,-176.040,9.172,148.709
C06217=1175.588,403.802,-84.659,-176.040,9.170,148.709
C06218=1175.592,403.554,-84.623,-176.040,9.168,148.708
C06219=1175.596,403.307,-84.587,-176.039,9.166,148.708
C06220=1175.600,403.059,-84.550,-176.039,9.164,148.707
C06221=1175.603,402.812,-84.515,-176.039,9.161,148.706
C06222=1175.608,402.565,-84.480,-176.038,9.159,148.706
C06223=1175.612,402.318,-84.443,-176.039,9.157,148.705
C06224=1175.615,402.070,-84.407,-176.038,9.154,148.704
C06225=1175.620,401.823,-84.371,-176.038,9.152,148.704
C06226=1175.623,401.575,-84.336,-176.038,9.150,148.703
C06227=1175.627,401.328,-84.299,-176.038,9.148,148.703
C06228=1175.631,401.080,-84.263,-176.038,9.145,148.702
C06229=1175.635,400.833,-84.228,-176.038,9.143,148.701
C06230=1175.639,400.585,-84.192,-176.038,9.140,148.701
C06231=1175.643,400.339,-84.156,-176.038,9.138,148.700
C06232=1175.647,400.091,-84.120,-176.037,9.136,148.699
C06233=1175.651,399.844,-84.084,-176.037,9.134,148.699
C06234=1175.655,399.596,-84.048,-176.037,9.131,148.698
C06235=1175.658,399.349,-84.012,-176.037,9.129,148.697
C06236=1175.663,399.101,-83.976,-176.037,9.126,148.697
C06237=1175.666,398.854,-83.940,-176.037,9.124,148.696
C06238=1175.670,398.606,-83.905,-176.037,9.121,148.695
C06239=1175.674,398.359,-83.868,-176.037,9.119,148.695
C06240=1175.678,398.112,-83.833,-176.036,9.116,148.694
C06241=1175.682,397.865,-83.797,-176.037,9.114,148.693
C06242=1175.686,397.617,-83.761,-176.037,9.111,148.693
C06243=1175.690,397.370,-83.726,-176.036,9.109,148.692
C06244=1175.693,397.123,-83.689,-176.036,9.106,148.691
C06245=1175.698,396.875,-83.653,-176.037,9.104,148.691
C06246=1175.702,396.627,-83.618,-176.036,9.101,148.690
C06247=1175.706,396.381,-83.582,-176.036,9.099,148.689
C06248=1175.710,396.133,-83.546,-176.036,9.096,148.689
C06249=1175.714,395.885,-83.511,-176.036,9.094,148.688
C06250=1175.717,395.638,-83.474,-176.036,9.091,148.687
C06251=1175.722,395.391,-83.438,-176.036,9.089,148.687
C06252=1175.725,395.143,-83.403,-176.036,9.086,148.686
C06253=1175.729,394.896,-83.367,-176.036,9.084,148.685
C06254=1175.734,394.648,-83.331,-176.036,9.081,148.685
C06255=1175.738,394.401,-83.296,-176.036,9.078,148.684
C06256=1175.741,394.154,-83.260,-176.036,9.076,148.683
C06257=1175.745,393.907,-83.224,-176.036,9.073,148.682
C06258=1175.749,393.659,-83.188,-176.036,9.071,148.682
C06259=1175.753,393.411,-83.152,-176.037,9.067,148.681
C06260=1175.757,393.165,-83.117,-176.036,9.065,148.680
C06261=1175.761,392.917,-83.081,-176.036,9.062,148.680
C06262=1175.765,392.669,-83.046,-176.037,9.059,148.679
C06263=1175.769,392.422,-83.010,-176.037,9.056,148.678
C06264=1175.773,392.137,-82.968,-176.037,9.053,148.678
C06265=1175.777,391.853,-82.928,-176.037,9.051,148.677
C06266=1175.783,391.569,-82.886,-176.037,9.047,148.676
C06267=1175.787,391.284,-82.846,-176.038,9.043,148.675
C06268=1175.791,391.036,-82.810,-176.037,9.041,148.674
C06269=1175.795,390.789,-82.774,-176.038,9.038,148.674
C06270=1175.798,390.542,-82.738,-176.038,9.035,148.673
C06271=1175.802,390.294,-82.703,-176.039,9.032,148.672
C06272=1175.807,390.047,-82.667,-176.039,9.030,148.672
C06273=1175.810,389.800,-82.631,-176.039,9.026,148.671
C06274=1175.814,389.552,-82.596,-176.039,9.024,148.670
C06275=1175.818,389.305,-82.560,-176.040,9.020,148.670
C06276=1175.822,389.057,-82.524,-176.040,9.018,148.669
C06277=1175.826,388.810,-82.489,-176.040,9.015,148.668
C06278=1175.830,388.563,-82.453,-176.041,9.011,148.668
C06279=1175.834,388.315,-82.418,-176.041,9.009,148.667
C06280=1175.837,388.068,-82.382,-176.041,9.005,148.666
C06281=1175.842,387.820,-82.346,-176.042,9.002,148.666
C06282=1175.846,387.573,-82.311,-176.042,9.000,148.665
C06283=1175.850,387.326,-82.275,-176.043,8.997,148.664
C06284=1175.853,387.078,-82.240,-176.043,8.993,148.664
C06285=1175.857,386.831,-82.204,-176.043,8.990,148.663
C06286=1175.861,386.583,-82.169,-176.044,8.988,148.662
C06287=1175.866,386.336,-82.133,-176.044,8.984,148.661
C06288=1175.869,386.089,-82.097,-176.045,8.981,148.661
C06289=1175.873,385.840,-82.062,-176.045,8.978,148.660
C06290=1175.877,385.593,-82.027,-176.046,8.975,148.660
C06291=1175.881,385.346,-81.992,-176.047,8.971,148.659
C06292=1175.885,385.099,-81.956,-176.047,8.968,148.658
C06293=1175.889,384.851,-81.920,-176.048,8.965,148.658
C06294=1175.893,384.603,-81.884,-176.049,8.962,148.657
C06295=1175.897,384.356,-81.849,-176.050,8.959,148.656
C06296=1175.901,384.109,-81.814,-176.050,8.955,148.656
C06297=1175.905,383.861,-81.778,-176.051,8.952,148.655
C06298=1175.908,383.614,-81.743,-176.052,8.949,148.654
C06299=1175.913,383.367,-81.708,-176.052,8.946,148.654
C06300=1175.917,383.119,-81.672,-176.053,8.943,148.653
C06301=1175.921,382.871,-81.637,-176.054,8.940,148.652
C06302=1175.925,382.624,-81.601,-176.054,8.936,148.652
C06303=1175.929,382.377,-81.566,-176.055,8.933,148.651
C06304=1175.932,382.129,-81.530,-176.056,8.930,148.650
C06305=1175.936,381.881,-81.495,-176.057,8.926,148.650
C06306=1175.940,381.634,-81.460,-176.058,8.923,148.649
C06307=1175.944,381.387,-81.425,-176.058,8.920,148.648
C06308=1175.948,381.140,-81.389,-176.059,8.916,148.648
C06309=1175.952,380.891,-81.354,-176.060,8.913,148.647
C06310=1175.956,380.645,-81.319,-176.061,8.909,148.647
C06311=1175.960,380.397,-81.284,-176.062,8.906,148.646
C06312=1175.964,380.149,-81.247,-176.063,8.903,148.645
C06313=1175.969,379.902,-81.213,-176.064,8.899,148.645
C06314=1175.973,379.654,-81.177,-176.065,8.896,148.644
C06315=1175.976,379.407,-81.142,-176.066,8.893,148.644
C06316=1175.980,379.159,-81.106,-176.067,8.889,148.643
C06317=1175.984,378.912,-81.072,-176.068,8.886,148.642
C06318=1175.988,378.664,-81.036,-176.069,8.882,148.642
C06319=1175.992,378.417,-81.001,-176.070,8.879,148.641
C06320=1175.996,378.170,-80.966,-176.072,8.875,148.641
C06321=1176.000,377.922,-80.931,-176.072,8.872,148.640
C06322=1176.004,377.675,-80.895,-176.073,8.869,148.639
C06323=1176.008,377.427,-80.861,-176.075,8.865,148.639
C06324=1176.012,377.180,-80.825,-176.076,8.862,148.638
C06325=1176.016,376.931,-80.790,-176.077,8.858,148.638
C06326=1176.020,376.685,-80.755,-176.079,8.854,148.637
C06327=1176.024,376.437,-80.720,-176.080,8.851,148.636
C06328=1176.028,376.189,-80.685,-176.081,8.847,148.636
C06329=1176.032,375.942,-80.650,-176.082,8.844,148.635
C06330=1176.036,375.694,-80.615,-176.084,8.840,148.635
C06331=1176.040,375.448,-80.580,-176.085,8.837,148.634
C06332=1176.043,375.200,-80.545,-176.086,8.833,148.634
C06333=1176.047,374.952,-80.510,-176.088,8.830,148.633
C06334=1176.051,374.705,-80.475,-176.088,8.827,148.633
C06335=1176.055,374.457,-80.440,-176.090,8.823,148.632
C06336=1176.059,374.210,-80.404,-176.092,8.819,148.632
C06337=1176.064,373.962,-80.370,-176.093,8.815,148.631
C06338=1176.067,373.715,-80.334,-176.094,8.812,148.630
C06339=1176.072,373.467,-80.300,-176.096,8.809,148.630
C06340=1176.076,373.219,-80.265,-176.097,8.805,148.629
C06341=1176.079,372.972,-80.230,-176.098,8.802,148.629
C06342=1176.083,372.725,-80.196,-176.100,8.798,148.628
C06343=1176.087,372.477,-80.160,-176.102,8.794,148.628
C06344=1176.092,372.230,-80.125,-176.103,8.790,148.627
C06345=1176.095,371.982,-80.090,-176.105,8.787,148.627
C06346=1176.100,371.735,-80.055,-176.106,8.784,148.626
C06347=1176.103,371.487,-80.021,-176.108,8.780,148.626
C06348=1176.107,371.239,-79.986,-176.109,8.776,148.625
C06349=1176.111,370.992,-79.951,-176.111,8.773,148.625
C06350=1176.115,370.744,-79.916,-176.113,8.769,148.624
C06351=1176.119,370.497,-79.881,-176.114,8.765,148.624
C06352=1176.123,370.249,-79.847,-176.116,8.761,148.623
C06353=1176.127,370.002,-79.813,-176.117,8.759,148.623
C06354=1176.131,369.754,-79.777,-176.119,8.755,148.622
C06355=1176.136,369.507,-79.742,-176.120,8.751,148.622
C06356=1176.139,369.259,-79.708,-176.122,8.748,148.621
C06357=1176.143,369.011,-79.673,-176.124,8.744,148.621
C06358=1176.147,368.764,-79.638,-176.126,8.740,148.620
C06359=1176.151,368.516,-79.603,-176.128,8.737,148.620
C06360=1176.156,368.269,-79.569,-176.129,8.733,148.619
C06361=1176.159,368.021,-79.535,-176.131,8.729,148.619
C06362=1176.163,367.774,-79.500,-176.133,8.726,148.619
C06363=1176.167,367.526,-79.465,-176.135,8.722,148.618
C06364=1176.171,367.279,-79.431,-176.136,8.718,148.618
C06365=1176.175,367.031,-79.396,-176.138,8.715,148.617
C06366=1176.179,366.783,-79.362,-176.140,8.711,148.617
C06367=1176.183,366.535,-79.327,-176.142,8.708,148.616
C06368=1176.187,366.254,-79.288,-176.144,8.704,148.616
C06369=1176.192,365.972,-79.248,-176.146,8.699,148.616
C06370=1176.197,365.691,-79.209,-176.149,8.695,148.615
C06371=1176.201,365.409,-79.170,-176.150,8.691,148.615
C06372=1176.205,365.161,-79.135,-176.152,8.688,148.614
C06373=1176.209,364.913,-79.100,-176.154,8.684,148.614
C06374=1176.213,364.666,-79.067,-176.156,8.681,148.613
C06375=1176.218,364.418,-79.032,-176.158,8.677,148.613
C06376=1176.221,364.171,-78.998,-176.161,8.673,148.613
C06377=1176.225,363.923,-78.963,-176.162,8.669,148.612
C06378=1176.229,363.675,-78.929,-176.164,8.666,148.612
C06379=1176.233,363.428,-78.895,-176.166,8.662,148.611
C06380=1176.237,363.180,-78.860,-176.168,8.659,148.611
C06381=1176.241,362.933,-78.826,-176.170,8.655,148.611
C06382=1176.245,362.685,-78.791,-176.172,8.651,148.610
C06383=1176.249,362.438,-78.757,-176.174,8.648,148.610
C06384=1176.253,362.190,-78.723,-176.176,8.645,148.610
C06385=1176.257,361.942,-78.689,-176.178,8.641,148.609
C06386=1176.261,361.695,-78.654,-176.181,8.637,148.609
C06387=1176.264,361.447,-78.620,-176.183,8.633,148.608
C06388=1176.269,361.199,-78.586,-176.184,8.630,148.608
C06389=1176.273,360.952,-78.552,-176.187,8.626,148.608
C06390=1176.277,360.704,-78.517,-176.189,8.623,148.607
C06391=1176.281,360.457,-78.484,-176.191,8.619,148.607
C06392=1176.286,360.209,-78.449,-176.193,8.616,148.607
C06393=1176.289,359.961,-78.415,-176.195,8.612,148.606
C06394=1176.294,359.713,-78.381,-176.197,8.608,148.606
C06395=1176.298,359.466,-78.347,-176.200,8.605,148.606
C06396=1176.301,359.218,-78.312,-176.201,8.601,148.605
C06397=1176.305,358.971,-78.278,-176.204,8.598,148.605
C06398=1176.309,358.723,-78.245,-176.205,8.594,148.605
C06399=1176.313,358.475,-78.210,-176.208,8.590,148.604
C06400=1176.317,358.228,-78.177,-176.211,8.587,148.604
C06401=1176.322,357.981,-78.142,-176.212,8.583,148.604
C06402=1176.325,357.732,-78.109,-176.215,8.580,148.604
C06403=1176.329,357.485,-78.075,-176.217,8.576,148.603
C06404=1176.334,357.238,-78.040,-176.219,8.573,148.603
C06405=1176.337,356.989,-78.007,-176.222,8.569,148.603
C06406=1176.342,356.742,-77.972,-176.223,8.565,148.602
C06407=1176.346,356.495,-77.938,-176.226,8.562,148.602
C06408=1176.349,356.246,-77.905,-176.228,8.558,148.602
C06409=1176.354,355.999,-77.870,-176.230,8.555,148.601
C06410=1176.358,355.751,-77.837,-176.232,8.552,148.601
C06411=1176.362,355.504,-77.803,-176.235,8.547,148.601
C06412=1176.366,355.255,-77.769,-176.237,8.544,148.600
C06413=1176.370,355.008,-77.735,-176.239,8.540,148.600
C06414=1176.374,354.761,-77.702,-176.241,8.537,148.600
C06415=1176.378,354.513,-77.668,-176.244,8.534,148.600
C06416=1176.382,354.265,-77.634,-176.245,8.530,148.599
C06417=1176.386,354.018,-77.600,-176.248,8.526,148.599
C06418=1176.390,353.770,-77.567,-176.251,8.523,148.599
C06419=1176.395,353.522,-77.533,-176.253,8.520,148.599
C06420=1176.398,353.274,-77.499,-176.255,8.516,148.598
C06421=1176.402,353.027,-77.465,-176.257,8.513,148.598
C06422=1176.406,352.779,-77.432,-176.259,8.509,148.598
C06423=1176.411,352.532,-77.398,-176.262,8.505,148.598
C06424=1176.415,352.284,-77.365,-176.264,8.502,148.597
C06425=1176.418,352.036,-77.331,-176.266,8.498,148.597
C06426=1176.422,351.788,-77.297,-176.268,8.495,148.597
C06427=1176.426,351.541,-77.264,-176.271,8.492,148.596
C06428=1176.431,351.293,-77.230,-176.273,8.488,148.596
C06429=1176.435,351.046,-77.196,-176.275,8.485,148.596
C06430=1176.439,350.797,-77.163,-176.278,8.481,148.596
C06431=1176.443,350.549,-77.130,-176.280,8.477,148.595
C06432=1176.447,350.302,-77.096,-176.282,8.474,148.595
C06433=1176.451,350.055,-77.063,-176.284,8.471,148.595
C06434=1176.455,349.807,-77.030,-176.287,8.467,148.595
C06435=1176.460,349.559,-76.996,-176.289,8.464,148.594
C06436=1176.464,349.312,-76.962,-176.291,8.461,148.594
C06437=1176.467,349.063,-76.928,-176.294,8.457,148.594
C06438=1176.471,348.816,-76.895,-176.296,8.453,148.594
C06439=1176.475,348.568,-76.862,-176.299,8.450,148.594
C06440=1176.480,348.320,-76.829,-176.301,8.447,148.593
C06441=1176.483,348.073,-76.795,-176.303,8.443,148.593
C06442=1176.488,347.825,-76.762,-176.305,8.440,148.593
C06443=1176.492,347.578,-76.729,-176.307,8.436,148.592
C06444=1176.496,347.330,-76.696,-176.310,8.433,148.592
C06445=1176.500,347.082,-76.662,-176.312,8.430,148.592
C06446=1176.503,346.834,-76.629,-176.315,8.426,148.592
C06447=1176.508,346.586,-76.595,-176.317,8.422,148.592
C06448=1176.512,346.338,-76.562,-176.319,8.419,148.591
C06449=1176.517,346.090,-76.529,-176.321,8.416,148.591
C06450=1176.521,345.842,-76.496,-176.324,8.412,148.591
C06451=1176.525,345.595,-76.463,-176.326,8.409,148.591
C06452=1176.529,345.347,-76.429,-176.328,8.406,148.590
C06453=1176.533,345.099,-76.396,-176.331,8.403,148.590
C06454=1176.537,344.851,-76.363,-176.333,8.398,148.590
C06455=1176.541,344.604,-76.330,-176.336,8.395,148.590
C06456=1176.545,344.356,-76.297,-176.338,8.392,148.590
C06457=1176.549,344.109,-76.264,-176.340,8.388,148.589
C06458=1176.553,343.861,-76.231,-176.342,8.385,148.589
C06459=1176.557,343.613,-76.198,-176.345,8.382,148.589
C06460=1176.561,343.365,-76.165,-176.347,8.379,148.589
C06461=1176.566,343.118,-76.132,-176.350,8.376,148.589
C06462=1176.570,342.870,-76.098,-176.352,8.372,148.588
C06463=1176.574,342.622,-76.065,-176.354,8.369,148.588
C06464=1176.578,342.375,-76.032,-176.357,8.365,148.588
C06465=1176.582,342.126,-76.000,-176.359,8.362,148.588
C06466=1176.587,341.878,-75.967,-176.362,8.358,148.588
C06467=1176.590,341.631,-75.934,-176.364,8.355,148.587
C06468=1176.594,341.383,-75.901,-176.366,8.352,148.587
C06469=1176.598,341.136,-75.868,-176.368,8.348,148.587
C06470=1176.603,340.887,-75.835,-176.371,8.345,148.587
C06471=1176.607,340.639,-75.802,-176.373,8.342,148.587
C06472=1176.611,340.361,-75.766,-176.376,8.338,148.586
C06473=1176.616,340.081,-75.728,-176.379,8.335,148.586
C06474=1176.621,339.802,-75.691,-176.381,8.330,148.586
C06475=1176.625,339.523,-75.654,-176.384,8.326,148.586
C06476=1176.629,339.275,-75.621,-176.387,8.323,148.586
C06477=1176.633,339.027,-75.588,-176.389,8.320,148.585
C06478=1176.637,338.780,-75.556,-176.392,8.317,148.585
C06479=1176.641,338.531,-75.523,-176.394,8.313,148.585
C06480=1176.646,338.284,-75.491,-176.396,8.310,148.585
C06481=1176.650,338.037,-75.457,-176.398,8.307,148.585
C06482=1176.654,337.789,-75.426,-176.401,8.304,148.585
C06483=1176.658,337.541,-75.392,-176.403,8.300,148.584
C06484=1176.662,337.292,-75.360,-176.406,8.297,148.584
C06485=1176.667,337.045,-75.327,-176.408,8.294,148.584
C06486=1176.670,336.797,-75.295,-176.410,8.291,148.584
C06487=1176.674,336.549,-75.262,-176.413,8.288,148.584
C06488=1176.679,336.301,-75.229,-176.416,8.283,148.584
C06489=1176.682,336.053,-75.197,-176.418,8.280,148.583
C06490=1176.687,335.806,-75.164,-176.420,8.277,148.583
C06491=1176.692,335.558,-75.132,-176.423,8.274,148.583
C06492=1176.695,335.310,-75.099,-176.425,8.270,148.583
C06493=1176.699,335.062,-75.067,-176.428,8.267,148.583
C06494=1176.703,334.814,-75.035,-176.430,8.264,148.582
C06495=1176.707,334.566,-75.002,-176.433,8.261,148.582
C06496=1176.712,334.318,-74.969,-176.435,8.258,148.582
C06497=1176.716,334.071,-74.937,-176.437,8.254,148.582
C06498=1176.720,333.823,-74.904,-176.439,8.251,148.582
C06499=1176.724,333.575,-74.873,-176.442,8.248,148.582
C06500=1176.728,333.327,-74.839,-176.444,8.245,148.582
C06501=1176.732,333.079,-74.807,-176.447,8.241,148.581
C06502=1176.736,332.832,-74.775,-176.449,8.238,148.581
C06503=1176.741,332.584,-74.742,-176.452,8.235,148.581
C06504=1176.745,332.336,-74.711,-176.454,8.232,148.581
C06505=1176.749,332.087,-74.678,-176.457,8.229,148.581
C06506=1176.752,331.840,-74.646,-176.459,8.225,148.581
C06507=1176.757,331.592,-74.613,-176.462,8.221,148.581
C06508=1176.761,331.344,-74.582,-176.464,8.218,148.581
C06509=1176.765,331.096,-74.548,-176.467,8.215,148.580
C06510=1176.769,330.848,-74.517,-176.469,8.212,148.580
C06511=1176.774,330.601,-74.485,-176.472,8.209,148.580
C06512=1176.778,330.353,-74.453,-176.474,8.205,148.580
C06513=1176.782,330.104,-74.420,-176.476,8.202,148.580
C06514=1176.786,329.857,-74.388,-176.479,8.199,148.580
C06515=1176.791,329.609,-74.356,-176.481,8.196,148.580
C06516=1176.794,329.361,-74.324,-176.483,8.192,148.579
C06517=1176.799,329.113,-74.291,-176.486,8.189,148.579
C06518=1176.802,328.865,-74.259,-176.488,8.186,148.579
C06519=1176.807,328.618,-74.228,-176.491,8.183,148.579
C06520=1176.811,328.369,-74.196,-176.493,8.180,148.579
C06521=1176.815,328.121,-74.164,-176.496,8.177,148.579
C06522=1176.819,327.873,-74.131,-176.498,8.174,148.579
C06523=1176.823,327.626,-74.099,-176.501,8.170,148.579
C06524=1176.827,327.378,-74.067,-176.503,8.167,148.578
C06525=1176.832,327.130,-74.035,-176.506,8.164,148.578
C06526=1176.836,326.882,-74.003,-176.508,8.161,148.578
C06527=1176.840,326.634,-73.971,-176.511,8.158,148.578
C06528=1176.844,326.386,-73.939,-176.513,8.154,148.578
C06529=1176.848,326.139,-73.908,-176.515,8.151,148.578
C06530=1176.852,325.891,-73.876,-176.518,8.148,148.578
C06531=1176.856,325.642,-73.843,-176.520,8.145,148.578
C06532=1176.861,325.395,-73.812,-176.523,8.142,148.578
C06533=1176.864,325.147,-73.780,-176.525,8.138,148.577
C06534=1176.869,324.898,-73.748,-176.528,8.135,148.577
C06535=1176.874,324.651,-73.717,-176.530,8.132,148.577
C06536=1176.877,324.403,-73.685,-176.533,8.129,148.577
C06537=1176.881,324.154,-73.653,-176.535,8.126,148.577
C06538=1176.886,323.907,-73.621,-176.537,8.123,148.577
C06539=1176.890,323.659,-73.589,-176.540,8.120,148.577
C06540=1176.894,323.411,-73.558,-176.542,8.116,148.577
C06541=1176.898,323.163,-73.527,-176.545,8.113,148.577
C06542=1176.902,322.914,-73.494,-176.547,8.110,148.576
C06543=1176.907,322.667,-73.463,-176.550,8.107,148.576
C06544=1176.910,322.419,-73.431,-176.552,8.104,148.576
C06545=1176.915,322.172,-73.399,-176.555,8.101,148.576
C06546=1176.919,321.923,-73.368,-176.557,8.097,148.576
C06547=1176.923,321.675,-73.336,-176.560,8.094,148.576
C06548=1176.928,321.427,-73.304,-176.562,8.091,148.576
C06549=1176.931,321.179,-73.272,-176.565,8.088,148.576
C06550=1176.936,320.931,-73.242,-176.567,8.085,148.576
C06551=1176.940,320.683,-73.210,-176.570,8.082,148.576
C06552=1176.944,320.436,-73.178,-176.572,8.078,148.575
C06553=1176.948,320.187,-73.147,-176.575,8.075,148.575
C06554=1176.952,319.939,-73.115,-176.577,8.072,148.575
C06555=1176.957,319.692,-73.083,-176.580,8.069,148.575
C06556=1176.961,319.443,-73.052,-176.582,8.066,148.575
C06557=1176.965,319.196,-73.021,-176.585,8.063,148.575
C06558=1176.969,318.947,-72.989,-176.587,8.060,148.575
C06559=1176.973,318.700,-72.958,-176.590,8.057,148.575
C06560=1176.977,318.452,-72.926,-176.592,8.053,148.575
C06561=1176.982,318.204,-72.895,-176.595,8.050,148.575
C06562=1176.985,317.956,-72.864,-176.598,8.047,148.575
C06563=1176.990,317.708,-72.833,-176.600,8.044,148.574
C06564=1176.994,317.460,-72.801,-176.603,8.041,148.574
C06565=1176.998,317.212,-72.770,-176.605,8.038,148.574
C06566=1177.002,316.964,-72.738,-176.608,8.035,148.574
C06567=1177.007,316.716,-72.708,-176.610,8.031,148.574
C06568=1177.010,316.468,-72.676,-176.613,8.028,148.574
C06569=1177.015,316.220,-72.645,-176.615,8.025,148.574
C06570=1177.019,315.972,-72.613,-176.618,8.022,148.574
C06571=1177.023,315.724,-72.582,-176.621,8.019,148.574
C06572=1177.027,315.475,-72.551,-176.623,8.016,148.574
C06573=1177.031,315.228,-72.520,-176.626,8.013,148.574
C06574=1177.036,314.980,-72.489,-176.628,8.009,148.574
C06575=1177.040,314.732,-72.457,-176.631,8.007,148.574
C06576=1177.045,314.454,-72.423,-176.633,8.004,148.574
C06577=1177.049,314.178,-72.388,-176.636,7.999,148.573
C06578=1177.054,313.901,-72.353,-176.639,7.996,148.573
C06579=1177.059,313.624,-72.319,-176.642,7.993,148.573
C06580=1177.063,313.376,-72.287,-176.644,7.989,148.573
C06581=1177.068,313.129,-72.257,-176.647,7.986,148.573
C06582=1177.072,312.880,-72.225,-176.649,7.983,148.573
C06583=1177.076,312.633,-72.194,-176.652,7.981,148.573
C06584=1177.079,312.384,-72.163,-176.654,7.978,148.573
C06585=1177.084,312.136,-72.133,-176.657,7.975,148.573
C06586=1177.088,311.888,-72.102,-176.659,7.972,148.573
C06587=1177.092,311.640,-72.071,-176.662,7.968,148.573
C06588=1177.097,311.392,-72.039,-176.664,7.965,148.573
C06589=1177.101,311.144,-72.009,-176.667,7.962,148.573
C06590=1177.105,310.896,-71.978,-176.669,7.959,148.572
C06591=1177.109,310.648,-71.947,-176.672,7.956,148.572
C06592=1177.114,310.400,-71.916,-176.675,7.953,148.572
C06593=1177.118,310.151,-71.885,-176.677,7.950,148.572
C06594=1177.122,309.903,-71.855,-176.680,7.947,148.572
C06595=1177.126,309.656,-71.824,-176.682,7.944,148.572
C06596=1177.130,309.408,-71.793,-176.685,7.940,148.572
C06597=1177.135,309.160,-71.762,-176.687,7.937,148.572
C06598=1177.139,308.912,-71.731,-176.690,7.934,148.572
C06599=1177.142,308.663,-71.700,-176.692,7.931,148.572
C06600=1177.147,308.416,-71.670,-176.695,7.928,148.572
C06601=1177.152,308.168,-71.639,-176.698,7.925,148.572
C06602=1177.156,307.919,-71.608,-176.700,7.923,148.572
C06603=1177.160,307.671,-71.578,-176.702,7.920,148.572
C06604=1177.164,307.423,-71.547,-176.705,7.917,148.572
C06605=1177.169,307.175,-71.516,-176.707,7.913,148.572
C06606=1177.172,306.927,-71.486,-176.710,7.910,148.572
C06607=1177.177,306.679,-71.455,-176.713,7.907,148.572
C06608=1177.181,306.431,-71.424,-176.715,7.904,148.572
C06609=1177.185,306.183,-71.394,-176.718,7.901,148.572
C06610=1177.190,305.934,-71.363,-176.720,7.898,148.572
C06611=1177.194,305.686,-71.333,-176.723,7.895,148.571
C06612=1177.198,305.439,-71.303,-176.725,7.892,148.571
C06613=1177.203,305.191,-71.272,-176.728,7.889,148.571
C06614=1177.207,304.942,-71.241,-176.731,7.886,148.571
C06615=1177.211,304.694,-71.210,-176.733,7.883,148.571
C06616=1177.215,304.446,-71.180,-176.735,7.880,148.571
C06617=1177.219,304.198,-71.150,-176.738,7.877,148.571
C06618=1177.223,303.949,-71.119,-176.740,7.874,148.571
C06619=1177.228,303.701,-71.088,-176.743,7.871,148.571
C06620=1177.232,303.454,-71.058,-176.746,7.868,148.571
C06621=1177.237,303.205,-71.028,-176.749,7.865,148.571
C06622=1177.241,302.958,-70.998,-176.751,7.862,148.571
C06623=1177.245,302.709,-70.967,-176.754,7.859,148.571
C06624=1177.248,302.461,-70.937,-176.756,7.856,148.571
C06625=1177.253,302.213,-70.907,-176.759,7.853,148.571
C06626=1177.257,301.965,-70.876,-176.761,7.850,148.571
C06627=1177.262,301.717,-70.846,-176.763,7.847,148.571
C06628=1177.266,301.469,-70.816,-176.766,7.844,148.571
C06629=1177.270,301.220,-70.785,-176.768,7.841,148.571
C06630=1177.274,300.973,-70.755,-176.771,7.838,148.571
C06631=1177.279,300.724,-70.725,-176.774,7.835,148.571
C06632=1177.283,300.476,-70.695,-176.777,7.832,148.571
C06633=1177.288,300.228,-70.665,-176.779,7.829,148.571
C06634=1177.292,299.980,-70.635,-176.782,7.826,148.571
C06635=1177.296,299.732,-70.604,-176.784,7.823,148.571
C06636=1177.300,299.484,-70.574,-176.787,7.820,148.571
C06637=1177.304,299.235,-70.543,-176.789,7.818,148.571
C06638=1177.309,298.987,-70.514,-176.792,7.814,148.571
C06639=1177.312,298.739,-70.484,-176.794,7.811,148.571
C06640=1177.317,298.491,-70.454,-176.797,7.808,148.571
C06641=1177.321,298.243,-70.423,-176.800,7.805,148.571
C06642=1177.325,297.995,-70.394,-176.802,7.802,148.571
C06643=1177.330,297.747,-70.363,-176.805,7.799,148.571
C06644=1177.334,297.499,-70.334,-176.807,7.796,148.571
C06645=1177.339,297.251,-70.303,-176.810,7.793,148.571
C06646=1177.343,297.002,-70.273,-176.812,7.791,148.571
C06647=1177.347,296.754,-70.244,-176.815,7.788,148.571
C06648=1177.351,296.505,-70.213,-176.817,7.785,148.571
C06649=1177.355,296.257,-70.183,-176.820,7.782,148.571
C06650=1177.359,296.009,-70.153,-176.823,7.779,148.571
C06651=1177.363,295.761,-70.124,-176.826,7.776,148.571
C06652=1177.368,295.513,-70.094,-176.828,7.772,148.570
C06653=1177.372,295.265,-70.064,-176.831,7.769,148.570
C06654=1177.376,295.017,-70.034,-176.833,7.767,148.571
C06655=1177.381,294.768,-70.004,-176.835,7.764,148.571
C06656=1177.385,294.520,-69.974,-176.838,7.761,148.571
C06657=1177.389,294.272,-69.944,-176.840,7.758,148.570
C06658=1177.394,294.024,-69.915,-176.843,7.755,148.570
C06659=1177.398,293.776,-69.886,-176.846,7.752,148.570
C06660=1177.402,293.528,-69.855,-176.849,7.749,148.570
C06661=1177.407,293.279,-69.825,-176.851,7.746,148.571
C06662=1177.411,293.031,-69.796,-176.853,7.744,148.571
C06663=1177.415,292.783,-69.766,-176.856,7.741,148.570
C06664=1177.419,292.535,-69.737,-176.858,7.738,148.570
C06665=1177.424,292.287,-69.706,-176.861,7.735,148.570
C06666=1177.428,292.038,-69.677,-176.864,7.732,148.571
C06667=1177.432,291.790,-69.647,-176.867,7.729,148.571
C06668=1177.436,291.542,-69.618,-176.869,7.726,148.571
C06669=1177.440,291.294,-69.588,-176.871,7.723,148.570
C06670=1177.445,291.045,-69.559,-176.874,7.720,148.570
C06671=1177.450,290.797,-69.529,-176.877,7.717,148.570
C06672=1177.454,290.549,-69.499,-176.879,7.714,148.571
C06673=1177.458,290.301,-69.469,-176.882,7.711,148.571
C06674=1177.462,290.053,-69.440,-176.885,7.708,148.571
C06675=1177.467,289.805,-69.411,-176.887,7.706,148.571
C06676=1177.471,289.557,-69.381,-176.889,7.703,148.570
C06677=1177.475,289.309,-69.352,-176.892,7.700,148.571
C06678=1177.479,289.060,-69.322,-176.895,7.697,148.571
C06679=1177.483,288.812,-69.293,-176.897,7.694,148.571
C06680=1177.488,288.537,-69.260,-176.900,7.691,148.571
C06681=1177.493,288.263,-69.227,-176.903,7.688,148.571
C06682=1177.498,287.987,-69.195,-176.906,7.684,148.571
C06683=1177.503,287.712,-69.163,-176.909,7.681,148.571
C06684=1177.507,287.465,-69.134,-176.912,7.678,148.571
C06685=1177.512,287.216,-69.104,-176.914,7.676,148.571
C06686=1177.516,286.968,-69.075,-176.917,7.673,148.571
C06687=1177.520,286.720,-69.045,-176.919,7.670,148.571
C06688=1177.524,286.471,-69.016,-176.922,7.667,148.571
C06689=1177.528,286.223,-68.986,-176.924,7.664,148.571
C06690=1177.532,285.975,-68.957,-176.927,7.661,148.571
C06691=1177.538,285.727,-68.929,-176.929,7.659,148.571
C06692=1177.542,285.478,-68.899,-176.932,7.656,148.571
C06693=1177.546,285.230,-68.870,-176.935,7.653,148.571
C06694=1177.550,284.982,-68.840,-176.937,7.650,148.571
C06695=1177.554,284.734,-68.811,-176.940,7.647,148.571
C06696=1177.558,284.485,-68.783,-176.943,7.644,148.571
C06697=1177.563,284.238,-68.754,-176.945,7.642,148.571
C06698=1177.567,283.989,-68.724,-176.948,7.639,148.571
C06699=1177.571,283.741,-68.695,-176.950,7.636,148.571
C06700=1177.576,283.492,-68.666,-176.953,7.632,148.571
C06701=1177.580,283.244,-68.636,-176.955,7.629,148.571
C06702=1177.585,282.996,-68.607,-176.958,7.627,148.571
C06703=1177.589,282.747,-68.579,-176.960,7.624,148.571
C06704=1177.593,282.499,-68.550,-176.963,7.621,148.571
C06705=1177.597,282.251,-68.520,-176.966,7.618,148.571
C06706=1177.602,282.003,-68.492,-176.969,7.615,148.571
C06707=1177.606,281.755,-68.462,-176.971,7.613,148.571
C06708=1177.610,281.506,-68.433,-176.973,7.610,148.571
C06709=1177.615,281.258,-68.404,-176.976,7.607,148.571
C06710=1177.619,281.010,-68.376,-176.979,7.604,148.571
C06711=1177.623,280.761,-68.347,-176.982,7.601,148.571
C06712=1177.627,280.513,-68.318,-176.984,7.599,148.572
C06713=1177.632,280.264,-68.289,-176.987,7.596,148.572
C06714=1177.637,280.017,-68.260,-176.989,7.593,148.572
C06715=1177.640,279.769,-68.231,-176.992,7.590,148.572
C06716=1177.645,279.520,-68.202,-176.995,7.587,148.572
C06717=1177.649,279.272,-68.173,-176.997,7.585,148.572
C06718=1177.654,279.023,-68.144,-177.000,7.582,148.572
C06719=1177.658,278.775,-68.116,-177.002,7.579,148.572
C06720=1177.662,278.527,-68.087,-177.005,7.576,148.572
C06721=1177.667,278.278,-68.058,-177.007,7.573,148.572
C06722=1177.670,278.030,-68.030,-177.010,7.570,148.572
C06723=1177.675,277.781,-68.001,-177.012,7.568,148.572
C06724=1177.680,277.534,-67.972,-177.015,7.565,148.572
C06725=1177.683,277.285,-67.944,-177.018,7.562,148.572
C06726=1177.688,277.036,-67.915,-177.020,7.559,148.572
C06727=1177.693,276.789,-67.886,-177.023,7.556,148.572
C06728=1177.696,276.540,-67.858,-177.025,7.553,148.572
C06729=1177.701,276.291,-67.829,-177.028,7.550,148.572
C06730=1177.706,276.044,-67.800,-177.030,7.548,148.572
C06731=1177.709,275.795,-67.772,-177.033,7.545,148.572
C06732=1177.714,275.546,-67.743,-177.036,7.542,148.572
C06733=1177.718,275.299,-67.714,-177.039,7.539,148.572
C06734=1177.722,275.050,-67.686,-177.041,7.537,148.572
C06735=1177.728,274.802,-67.657,-177.043,7.534,148.572
C06736=1177.731,274.554,-67.628,-177.046,7.531,148.572
C06737=1177.735,274.305,-67.600,-177.049,7.528,148.573
C06738=1177.740,274.057,-67.572,-177.051,7.526,148.573
C06739=1177.744,273.808,-67.543,-177.054,7.523,148.573
C06740=1177.749,273.561,-67.515,-177.057,7.520,148.573
C06741=1177.753,273.312,-67.486,-177.060,7.518,148.573
C06742=1177.757,273.063,-67.457,-177.062,7.515,148.573
C06743=1177.762,272.816,-67.429,-177.065,7.512,148.573
C06744=1177.766,272.567,-67.401,-177.067,7.509,148.573
C06745=1177.770,272.319,-67.373,-177.070,7.506,148.573
C06746=1177.775,272.070,-67.344,-177.072,7.504,148.573
C06747=1177.779,271.822,-67.316,-177.075,7.501,148.573
C06748=1177.783,271.574,-67.287,-177.078,7.498,148.573
C06749=1177.787,271.325,-67.259,-177.080,7.495,148.573
C06750=1177.792,271.077,-67.230,-177.083,7.493,148.573
C06751=1177.796,270.828,-67.202,-177.085,7.490,148.574
C06752=1177.800,270.581,-67.174,-177.088,7.487,148.574
C06753=1177.805,270.332,-67.146,-177.091,7.484,148.574
C06754=1177.809,270.084,-67.118,-177.093,7.482,148.574
C06755=1177.814,269.835,-67.089,-177.096,7.479,148.574
C06756=1177.818,269.587,-67.061,-177.098,7.476,148.574
C06757=1177.823,269.338,-67.033,-177.101,7.474,148.574
C06758=1177.827,269.090,-67.005,-177.103,7.471,148.574
C06759=1177.831,268.842,-66.977,-177.106,7.468,148.574
C06760=1177.836,268.594,-66.948,-177.109,7.465,148.574
C06761=1177.840,268.345,-66.920,-177.112,7.463,148.574
C06762=1177.845,268.097,-66.892,-177.114,7.460,148.574
C06763=1177.849,267.848,-66.864,-177.117,7.457,148.574
C06764=1177.853,267.600,-66.837,-177.119,7.455,148.575
C06765=1177.858,267.351,-66.808,-177.122,7.452,148.575
C06766=1177.862,267.103,-66.780,-177.125,7.449,148.575
C06767=1177.866,266.855,-66.752,-177.127,7.446,148.575
C06768=1177.871,266.606,-66.724,-177.130,7.444,148.575
C06769=1177.875,266.358,-66.696,-177.132,7.441,148.575
C06770=1177.879,266.109,-66.668,-177.135,7.438,148.575
C06771=1177.883,265.861,-66.641,-177.138,7.436,148.575
C06772=1177.888,265.612,-66.612,-177.140,7.433,148.575
C06773=1177.892,265.364,-66.584,-177.143,7.430,148.575
C06774=1177.897,265.117,-66.556,-177.146,7.427,148.575
C06775=1177.901,264.867,-66.528,-177.148,7.425,148.575
C06776=1177.906,264.619,-66.501,-177.151,7.422,148.575
C06777=1177.910,264.371,-66.472,-177.154,7.419,148.575
C06778=1177.914,264.122,-66.445,-177.156,7.417,148.576
C06779=1177.919,263.874,-66.417,-177.158,7.414,148.576
C06780=1177.923,263.625,-66.389,-177.162,7.411,148.576
C06781=1177.927,263.377,-66.361,-177.164,7.409,148.576
C06782=1177.931,263.128,-66.334,-177.167,7.406,148.576
C06783=1177.936,262.880,-66.306,-177.169,7.403,148.576
C06784=1177.940,262.607,-66.275,-177.172,7.400,148.576
C06785=1177.946,262.334,-66.245,-177.175,7.397,148.576
C06786=1177.950,262.061,-66.214,-177.178,7.395,148.576
C06787=1177.956,261.788,-66.184,-177.181,7.392,148.576
C06788=1177.960,261.539,-66.157,-177.183,7.389,148.577
C06789=1177.964,261.291,-66.129,-177.186,7.387,148.577
C06790=1177.968,261.044,-66.101,-177.188,7.384,148.577
C06791=1177.972,260.794,-66.074,-177.192,7.381,148.577
C06792=1177.978,260.546,-66.045,-177.194,7.379,148.577
C06793=1177.982,260.298,-66.018,-177.196,7.376,148.577
C06794=1177.986,260.049,-65.990,-177.199,7.373,148.577
C06795=1177.991,259.801,-65.963,-177.201,7.371,148.577
C06796=1177.995,259.553,-65.935,-177.204,7.368,148.577
C06797=1177.999,259.304,-65.908,-177.207,7.365,148.578
C06798=1178.003,259.056,-65.880,-177.209,7.363,148.578
C06799=1178.008,258.807,-65.853,-177.212,7.360,148.578
C06800=1178.012,258.558,-65.825,-177.214,7.358,148.578
C06801=1178.016,258.310,-65.798,-177.217,7.355,148.578
C06802=1178.021,258.062,-65.771,-177.220,7.352,148.578
C06803=1178.025,257.814,-65.743,-177.223,7.350,148.578
C06804=1178.030,257.565,-65.715,-177.225,7.347,148.578
C06805=1178.034,257.316,-65.688,-177.228,7.344,148.578
C06806=1178.039,257.068,-65.661,-177.230,7.342,148.578
C06807=1178.043,256.820,-65.633,-177.233,7.339,148.578
C06808=1178.047,256.570,-65.606,-177.236,7.336,148.579
C06809=1178.052,256.323,-65.578,-177.238,7.334,148.579
C06810=1178.056,256.074,-65.551,-177.241,7.331,148.579
C06811=1178.061,255.826,-65.524,-177.244,7.328,148.579
C06812=1178.065,255.577,-65.496,-177.246,7.326,148.579
C06813=1178.069,255.329,-65.469,-177.249,7.324,148.579
C06814=1178.074,255.080,-65.442,-177.251,7.321,148.579
C06815=1178.079,254.832,-65.415,-177.254,7.318,148.579
C06816=1178.083,254.584,-65.387,-177.257,7.315,148.580
C06817=1178.087,254.334,-65.360,-177.259,7.314,148.580
C06818=1178.092,254.086,-65.333,-177.262,7.311,148.580
C06819=1178.096,253.837,-65.305,-177.265,7.308,148.580
C06820=1178.101,253.589,-65.278,-177.267,7.306,148.580
C06821=1178.105,253.341,-65.251,-177.270,7.303,148.580
C06822=1178.109,253.092,-65.224,-177.272,7.301,148.580
C06823=1178.113,252.844,-65.197,-177.275,7.298,148.580
C06824=1178.118,252.595,-65.170,-177.278,7.295,148.581
C06825=1178.123,252.347,-65.143,-177.280,7.293,148.581
C06826=1178.127,252.098,-65.116,-177.283,7.290,148.581
C06827=1178.131,251.850,-65.089,-177.286,7.288,148.581
C06828=1178.136,251.602,-65.062,-177.288,7.285,148.581
C06829=1178.140,251.353,-65.034,-177.291,7.282,148.581
C06830=1178.144,251.104,-65.007,-177.294,7.280,148.581
C06831=1178.149,250.856,-64.980,-177.296,7.277,148.582
C06832=1178.154,250.607,-64.953,-177.299,7.275,148.582
C06833=1178.157,250.359,-64.926,-177.301,7.272,148.582
C06834=1178.162,250.111,-64.899,-177.305,7.269,148.582
C06835=1178.167,249.862,-64.872,-177.307,7.267,148.582
C06836=1178.171,249.614,-64.845,-177.309,7.264,148.582
C06837=1178.175,249.365,-64.818,-177.312,7.262,148.582
C06838=1178.179,249.116,-64.791,-177.315,7.259,148.582
C06839=1178.184,248.867,-64.765,-177.318,7.256,148.583
C06840=1178.189,248.619,-64.738,-177.320,7.254,148.583
C06841=1178.193,248.371,-64.711,-177.323,7.252,148.583
C06842=1178.198,248.122,-64.684,-177.325,7.250,148.583
C06843=1178.202,247.874,-64.657,-177.328,7.247,148.583
C06844=1178.206,247.625,-64.631,-177.331,7.245,148.583
C06845=1178.211,247.377,-64.604,-177.333,7.242,148.583
C06846=1178.216,247.128,-64.577,-177.336,7.239,148.584
C06847=1178.219,246.880,-64.550,-177.339,7.237,148.584
C06848=1178.224,246.631,-64.524,-177.341,7.234,148.584
C06849=1178.229,246.383,-64.497,-177.344,7.232,148.584
C06850=1178.233,246.134,-64.470,-177.346,7.229,148.584
C06851=1178.238,245.886,-64.443,-177.349,7.227,148.584
C06852=1178.242,245.637,-64.416,-177.352,7.224,148.584
C06853=1178.247,245.389,-64.390,-177.354,7.221,148.585
C06854=1178.251,245.140,-64.363,-177.357,7.219,148.585
C06855=1178.255,244.892,-64.337,-177.360,7.216,148.585
C06856=1178.259,244.643,-64.309,-177.362,7.214,148.585
C06857=1178.264,244.394,-64.283,-177.365,7.212,148.585
C06858=1178.268,244.145,-64.257,-177.367,7.209,148.585
C06859=1178.273,243.898,-64.230,-177.370,7.206,148.585
C06860=1178.278,243.649,-64.204,-177.373,7.205,148.586
C06861=1178.282,243.400,-64.177,-177.376,7.202,148.586
C06862=1178.286,243.152,-64.151,-177.378,7.199,148.586
C06863=1178.291,242.903,-64.124,-177.381,7.197,148.586
C06864=1178.295,242.655,-64.098,-177.384,7.194,148.586
C06865=1178.300,242.406,-64.071,-177.386,7.192,148.586
C06866=1178.304,242.158,-64.045,-177.389,7.189,148.587
C06867=1178.309,241.909,-64.018,-177.391,7.187,148.587
C06868=1178.313,241.660,-63.992,-177.394,7.184,148.587
C06869=1178.317,241.412,-63.965,-177.397,7.182,148.587
C06870=1178.321,241.164,-63.939,-177.399,7.179,148.587
C06871=1178.326,240.915,-63.912,-177.402,7.177,148.588
C06872=1178.330,240.666,-63.886,-177.405,7.174,148.588
C06873=1178.335,240.417,-63.860,-177.407,7.172,148.588
C06874=1178.339,240.169,-63.833,-177.410,7.170,148.588
C06875=1178.344,239.920,-63.807,-177.412,7.168,148.588
C06876=1178.348,239.672,-63.780,-177.415,7.165,148.588
C06877=1178.354,239.423,-63.754,-177.418,7.163,148.588
C06878=1178.357,239.175,-63.728,-177.420,7.160,148.589
C06879=1178.362,238.926,-63.702,-177.423,7.158,148.589
C06880=1178.367,238.677,-63.676,-177.426,7.155,148.589
C06881=1178.371,238.429,-63.649,-177.429,7.152,148.589
C06882=1178.376,238.180,-63.623,-177.431,7.150,148.589
C06883=1178.379,237.932,-63.596,-177.434,7.147,148.589
C06884=1178.384,237.683,-63.571,-177.437,7.145,148.590
C06885=1178.389,237.435,-63.545,-177.439,7.143,148.590
C06886=1178.393,237.186,-63.518,-177.442,7.140,148.590
C06887=1178.397,236.938,-63.492,-177.445,7.138,148.590
C06888=1178.402,236.666,-63.463,-177.447,7.136,148.590
C06889=1178.407,236.394,-63.435,-177.450,7.133,148.591
C06890=1178.412,236.123,-63.406,-177.453,7.130,148.591
C06891=1178.417,235.851,-63.378,-177.456,7.127,148.591
C06892=1178.422,235.602,-63.352,-177.458,7.125,148.591
C06893=1178.426,235.354,-63.326,-177.462,7.123,148.591
C06894=1178.430,235.105,-63.300,-177.464,7.120,148.591
C06895=1178.435,234.856,-63.274,-177.467,7.118,148.592
C06896=1178.439,234.608,-63.248,-177.469,7.116,148.592
C06897=1178.444,234.360,-63.222,-177.472,7.113,148.592
C06898=1178.448,234.111,-63.196,-177.475,7.111,148.592
C06899=1178.453,233.862,-63.170,-177.478,7.108,148.593
C06900=1178.457,233.613,-63.144,-177.480,7.106,148.593
C06901=1178.461,233.365,-63.118,-177.483,7.103,148.593
C06902=1178.466,233.116,-63.093,-177.485,7.101,148.593
C06903=1178.471,232.868,-63.066,-177.488,7.098,148.593
C06904=1178.475,232.619,-63.040,-177.491,7.097,148.593
C06905=1178.479,232.370,-63.014,-177.493,7.094,148.594
C06906=1178.484,232.122,-62.989,-177.496,7.092,148.594
C06907=1178.488,231.873,-62.963,-177.498,7.090,148.594
C06908=1178.493,231.624,-62.937,-177.502,7.087,148.594
C06909=1178.497,231.375,-62.911,-177.504,7.085,148.594
C06910=1178.502,231.127,-62.886,-177.507,7.082,148.595
C06911=1178.507,230.879,-62.860,-177.509,7.080,148.595
C06912=1178.511,230.630,-62.834,-177.512,7.077,148.595
C06913=1178.516,230.382,-62.809,-177.515,7.075,148.595
C06914=1178.520,230.133,-62.783,-177.517,7.072,148.595
C06915=1178.524,229.884,-62.757,-177.520,7.071,148.596
C06916=1178.529,229.635,-62.731,-177.523,7.068,148.596
C06917=1178.534,229.387,-62.706,-177.525,7.066,148.596
C06918=1178.538,229.138,-62.680,-177.528,7.064,148.596
C06919=1178.542,228.889,-62.654,-177.531,7.061,148.596
C06920=1178.547,228.641,-62.629,-177.533,7.059,148.596
C06921=1178.551,228.392,-62.603,-177.536,7.056,148.597
C06922=1178.556,228.144,-62.577,-177.538,7.054,148.597
C06923=1178.560,227.895,-62.552,-177.542,7.051,148.597
C06924=1178.565,227.647,-62.526,-177.544,7.049,148.597
C06925=1178.569,227.398,-62.500,-177.546,7.048,148.598
C06926=1178.574,227.150,-62.475,-177.549,7.045,148.598
C06927=1178.578,226.900,-62.450,-177.552,7.043,148.598
C06928=1178.582,226.651,-62.424,-177.555,7.040,148.598
C06929=1178.587,226.403,-62.399,-177.557,7.038,148.598
C06930=1178.591,226.155,-62.373,-177.560,7.035,148.599
C06931=1178.596,225.906,-62.347,-177.563,7.033,148.599
C06932=1178.600,225.658,-62.322,-177.565,7.031,148.599
C06933=1178.605,225.408,-62.297,-177.568,7.028,148.599
C06934=1178.610,225.160,-62.271,-177.571,7.027,148.600
C06935=1178.614,224.911,-62.246,-177.573,7.024,148.600
C06936=1178.618,224.663,-62.220,-177.576,7.022,148.600
C06937=1178.623,224.414,-62.195,-177.578,7.020,148.600
C06938=1178.628,224.165,-62.170,-177.581,7.017,148.600
C06939=1178.632,223.917,-62.144,-177.584,7.015,148.601
C06940=1178.637,223.668,-62.118,-177.587,7.012,148.601
C06941=1178.641,223.419,-62.093,-177.589,7.010,148.601
C06942=1178.645,223.171,-62.069,-177.592,7.008,148.601
C06943=1178.650,222.922,-62.043,-177.595,7.006,148.602
C06944=1178.655,222.673,-62.018,-177.597,7.004,148.602
C06945=1178.659,222.425,-61.992,-177.600,7.001,148.602
C06946=1178.664,222.176,-61.968,-177.603,6.999,148.602
C06947=1178.668,221.927,-61.942,-177.605,6.997,148.602
C06948=1178.672,221.678,-61.916,-177.608,6.994,148.603
C06949=1178.678,221.429,-61.892,-177.611,6.992,148.603
C06950=1178.681,221.181,-61.866,-177.614,6.990,148.603
C06951=1178.686,220.932,-61.842,-177.616,6.988,148.603
C06952=1178.690,220.683,-61.816,-177.619,6.986,148.604
C06953=1178.696,220.435,-61.791,-177.621,6.983,148.604
C06954=1178.700,220.186,-61.766,-177.624,6.981,148.604
C06955=1178.704,219.938,-61.741,-177.627,6.978,148.604
C06956=1178.708,219.689,-61.716,-177.629,6.976,148.604
C06957=1178.713,219.441,-61.690,-177.632,6.974,148.605
C06958=1178.718,219.191,-61.665,-177.635,6.971,148.605
C06959=1178.722,218.943,-61.641,-177.638,6.970,148.605
C06960=1178.726,218.694,-61.616,-177.640,6.968,148.605
C06961=1178.732,218.445,-61.591,-177.643,6.965,148.606
C06962=1178.736,218.196,-61.565,-177.646,6.963,148.606
C06963=1178.740,217.948,-61.541,-177.648,6.960,148.606
C06964=1178.744,217.699,-61.515,-177.651,6.958,148.606
C06965=1178.750,217.450,-61.491,-177.653,6.956,148.606
C06966=1178.754,217.201,-61.466,-177.656,6.954,148.607
C06967=1178.758,216.953,-61.441,-177.659,6.952,148.607
C06968=1178.763,216.705,-61.416,-177.661,6.950,148.607
C06969=1178.768,216.456,-61.390,-177.665,6.947,148.608
C06970=1178.772,216.207,-61.366,-177.667,6.945,148.608
C06971=1178.776,215.958,-61.341,-177.669,6.943,148.608
C06972=1178.781,215.710,-61.316,-177.673,6.941,148.608
C06973=1178.785,215.461,-61.291,-177.675,6.938,148.608
C06974=1178.790,215.212,-61.267,-177.677,6.937,148.609
C06975=1178.795,214.964,-61.243,-177.680,6.934,148.609
C06976=1178.799,214.715,-61.217,-177.683,6.932,148.609
C06977=1178.804,214.466,-61.192,-177.686,6.930,148.610
C06978=1178.808,214.217,-61.168,-177.688,6.927,148.610
C06979=1178.813,213.968,-61.143,-177.691,6.925,148.610
C06980=1178.818,213.720,-61.118,-177.694,6.923,148.610
C06981=1178.821,213.471,-61.093,-177.696,6.921,148.610
C06982=1178.827,213.222,-61.069,-177.699,6.919,148.611
C06983=1178.830,212.973,-61.044,-177.702,6.917,148.611
C06984=1178.836,212.724,-61.020,-177.704,6.914,148.611
C06985=1178.840,212.477,-60.995,-177.707,6.912,148.611
C06986=1178.844,212.227,-60.970,-177.709,6.910,148.612
C06987=1178.849,211.979,-60.946,-177.712,6.907,148.612
C06988=1178.854,211.730,-60.921,-177.715,6.906,148.612
C06989=1178.858,211.481,-60.896,-177.717,6.903,148.612
C06990=1178.863,211.232,-60.872,-177.721,6.901,148.613
C06991=1178.868,210.983,-60.847,-177.723,6.899,148.613
C06992=1178.872,210.713,-60.821,-177.726,6.896,148.613
C06993=1178.877,210.443,-60.794,-177.729,6.894,148.613
C06994=1178.882,210.173,-60.767,-177.732,6.892,148.614
C06995=1178.886,209.902,-60.740,-177.735,6.890,148.614
C06996=1178.892,209.653,-60.716,-177.738,6.887,148.614
C06997=1178.896,209.405,-60.691,-177.740,6.885,148.615
C06998=1178.900,209.155,-60.666,-177.743,6.883,148.615
C06999=1178.905,208.907,-60.642,-177.746,6.881,148.615
C07000=1178.909,208.658,-60.618,-177.748,6.879,148.615
C07001=1178.914,208.410,-60.594,-177.751,6.877,148.616
C07002=1178.918,208.160,-60.569,-177.754,6.874,148.616
C07003=1178.924,207.911,-60.545,-177.756,6.872,148.616
C07004=1178.928,207.663,-60.521,-177.759,6.870,148.616
C07005=1178.933,207.414,-60.496,-177.761,6.868,148.617
C07006=1178.937,207.165,-60.472,-177.764,6.866,148.617
C07007=1178.941,206.916,-60.448,-177.767,6.864,148.617
C07008=1178.946,206.668,-60.423,-177.770,6.862,148.618
C07009=1178.951,206.419,-60.399,-177.772,6.859,148.618
C07010=1178.955,206.170,-60.375,-177.775,6.857,148.618
C07011=1178.960,205.922,-60.350,-177.778,6.855,148.618
C07012=1178.964,205.672,-60.327,-177.780,6.854,148.619
C07013=1178.969,205.424,-60.303,-177.783,6.851,148.619
C07014=1178.973,205.175,-60.278,-177.786,6.849,148.619
C07015=1178.978,204.926,-60.254,-177.788,6.847,148.619
C07016=1178.982,204.678,-60.229,-177.791,6.844,148.620
C07017=1178.988,204.428,-60.206,-177.794,6.842,148.620
C07018=1178.992,204.180,-60.181,-177.796,6.841,148.620
C07019=1178.996,203.931,-60.157,-177.799,6.838,148.620
C07020=1179.001,203.682,-60.132,-177.802,6.836,148.621
C07021=1179.006,203.433,-60.109,-177.805,6.834,148.621
C07022=1179.010,203.185,-60.085,-177.807,6.832,148.621
C07023=1179.014,202.936,-60.061,-177.809,6.830,148.621
C07024=1179.019,202.687,-60.036,-177.813,6.827,148.622
C07025=1179.024,202.438,-60.012,-177.815,6.826,148.622
C07026=1179.028,202.189,-59.988,-177.817,6.824,148.622
C07027=1179.032,201.941,-59.964,-177.820,6.822,148.623
C07028=1179.037,201.692,-59.941,-177.823,6.819,148.623
C07029=1179.042,201.443,-59.916,-177.826,6.817,148.623
C07030=1179.046,201.194,-59.893,-177.828,6.815,148.623
C07031=1179.051,200.945,-59.868,-177.831,6.813,148.624
C07032=1179.055,200.697,-59.844,-177.834,6.811,148.624
C07033=1179.060,200.448,-59.821,-177.837,6.809,148.624
C07034=1179.065,200.199,-59.796,-177.839,6.807,148.625
C07035=1179.070,199.950,-59.773,-177.842,6.805,148.625
C07036=1179.074,199.702,-59.749,-177.845,6.802,148.625
C07037=1179.078,199.453,-59.725,-177.848,6.801,148.626
C07038=1179.083,199.204,-59.701,-177.850,6.799,148.626
C07039=1179.087,198.955,-59.677,-177.852,6.797,148.626
C07040=1179.092,198.706,-59.654,-177.856,6.794,148.626
C07041=1179.096,198.458,-59.630,-177.858,6.792,148.627
C07042=1179.102,198.208,-59.606,-177.861,6.790,148.627
C07043=1179.106,197.960,-59.582,-177.863,6.788,148.627
C07044=1179.111,197.711,-59.558,-177.866,6.786,148.627
C07045=1179.115,197.462,-59.535,-177.869,6.784,148.628
C07046=1179.120,197.213,-59.511,-177.871,6.782,148.628
C07047=1179.124,196.964,-59.487,-177.874,6.780,148.628
C07048=1179.129,196.716,-59.463,-177.877,6.778,148.629
C07049=1179.133,196.467,-59.440,-177.880,6.776,148.629
C07050=1179.138,196.218,-59.416,-177.882,6.774,148.629
C07051=1179.143,195.969,-59.393,-177.885,6.772,148.629
C07052=1179.147,195.720,-59.369,-177.887,6.770,148.630
C07053=1179.152,195.472,-59.345,-177.890,6.768,148.630
C07054=1179.156,195.223,-59.322,-177.893,6.766,148.630
C07055=1179.160,194.973,-59.298,-177.895,6.763,148.631
C07056=1179.165,194.725,-59.274,-177.898,6.762,148.631
C07057=1179.170,194.476,-59.251,-177.901,6.760,148.631
C07058=1179.174,194.227,-59.227,-177.903,6.758,148.632
C07059=1179.179,193.978,-59.203,-177.906,6.755,148.632
C07060=1179.183,193.729,-59.180,-177.909,6.753,148.632
C07061=1179.188,193.480,-59.156,-177.912,6.752,148.632
C07062=1179.193,193.231,-59.133,-177.914,6.750,148.633
C07063=1179.198,192.984,-59.109,-177.917,6.748,148.633
C07064=1179.202,192.734,-59.086,-177.920,6.745,148.633
C07065=1179.207,192.485,-59.063,-177.922,6.743,148.634
C07066=1179.212,192.236,-59.039,-177.925,6.742,148.634
C07067=1179.217,191.987,-59.016,-177.928,6.740,148.634
C07068=1179.221,191.739,-58.992,-177.930,6.738,148.635
C07069=1179.226,191.490,-58.969,-177.933,6.735,148.635
C07070=1179.230,191.241,-58.946,-177.936,6.733,148.635
C07071=1179.234,190.992,-58.922,-177.938,6.731,148.635
C07072=1179.239,190.743,-58.899,-177.941,6.730,148.636
C07073=1179.244,190.494,-58.876,-177.944,6.728,148.636
C07074=1179.248,190.245,-58.852,-177.946,6.726,148.636
C07075=1179.253,189.997,-58.828,-177.949,6.723,148.637
C07076=1179.258,189.748,-58.805,-177.952,6.721,148.637
C07077=1179.262,189.499,-58.782,-177.955,6.720,148.637
C07078=1179.266,189.250,-58.759,-177.957,6.718,148.638
C07079=1179.271,189.002,-58.736,-177.960,6.716,148.638
C07080=1179.276,188.753,-58.712,-177.962,6.714,148.638
C07081=1179.281,188.503,-58.689,-177.965,6.711,148.639
C07082=1179.286,188.254,-58.666,-177.968,6.709,148.639
C07083=1179.290,188.006,-58.643,-177.971,6.708,148.639
C07084=1179.294,187.757,-58.620,-177.973,6.706,148.640
C07085=1179.299,187.508,-58.596,-177.976,6.704,148.640
C07086=1179.304,187.259,-58.573,-177.978,6.702,148.640
C07087=1179.308,187.010,-58.550,-177.982,6.699,148.640
C07088=1179.313,186.762,-58.527,-177.984,6.698,148.641
C07089=1179.318,186.513,-58.504,-177.987,6.696,148.641
C07090=1179.322,186.264,-58.480,-177.990,6.694,148.641
C07091=1179.326,186.015,-58.458,-177.992,6.692,148.642
C07092=1179.331,185.766,-58.434,-177.994,6.690,148.642
C07093=1179.336,185.516,-58.412,-177.997,6.688,148.642
C07094=1179.341,185.268,-58.389,-178.000,6.686,148.643
C07095=1179.345,185.019,-58.366,-178.003,6.684,148.643
C07096=1179.351,184.749,-58.341,-178.006,6.682,148.643
C07097=1179.356,184.480,-58.316,-178.008,6.680,148.644
C07098=1179.360,184.211,-58.291,-178.012,6.678,148.644
C07099=1179.365,183.941,-58.266,-178.014,6.676,148.644
C07100=1179.370,183.692,-58.244,-178.017,6.674,148.645
C07101=1179.374,183.443,-58.220,-178.020,6.672,148.645
C07102=1179.379,183.194,-58.197,-178.023,6.670,148.645
C07103=1179.383,182.945,-58.174,-178.026,6.668,148.646
C07104=1179.388,182.696,-58.151,-178.028,6.666,148.646
C07105=1179.393,182.447,-58.128,-178.030,6.664,148.646
C07106=1179.397,182.198,-58.106,-178.033,6.662,148.647
C07107=1179.402,181.949,-58.082,-178.036,6.661,148.647
C07108=1179.407,181.701,-58.060,-178.038,6.659,148.647
C07109=1179.412,181.451,-58.037,-178.041,6.657,148.648
C07110=1179.416,181.202,-58.014,-178.044,6.654,148.648
C07111=1179.420,180.954,-57.991,-178.047,6.653,148.648
C07112=1179.426,180.705,-57.969,-178.049,6.651,148.649
C07113=1179.430,180.456,-57.946,-178.052,6.649,148.649
C07114=1179.435,180.207,-57.923,-178.055,6.647,148.649
C07115=1179.439,179.958,-57.901,-178.057,6.645,148.650
C07116=1179.444,179.709,-57.878,-178.060,6.643,148.650
C07117=1179.448,179.461,-57.855,-178.063,6.642,148.650
C07118=1179.453,179.211,-57.832,-178.065,6.640,148.651
C07119=1179.457,178.962,-57.810,-178.068,6.638,148.651
C07120=1179.463,178.713,-57.787,-178.071,6.636,148.651
C07121=1179.467,178.464,-57.765,-178.073,6.633,148.652
C07122=1179.471,178.215,-57.741,-178.076,6.632,148.652
C07123=1179.476,177.967,-57.719,-178.079,6.630,148.652
C07124=1179.481,177.718,-57.696,-178.081,6.628,148.653
C07125=1179.485,177.468,-57.674,-178.084,6.626,148.653
C07126=1179.490,177.220,-57.651,-178.087,6.625,148.653
C07127=1179.495,176.971,-57.629,-178.089,6.623,148.654
C07128=1179.499,176.722,-57.606,-178.092,6.621,148.654
C07129=1179.504,176.473,-57.584,-178.095,6.619,148.654
C07130=1179.508,176.224,-57.561,-178.097,6.617,148.655
C07131=1179.513,175.975,-57.539,-178.100,6.616,148.655
C07132=1179.518,175.727,-57.516,-178.102,6.614,148.655
C07133=1179.523,175.477,-57.494,-178.106,6.611,148.656
C07134=1179.527,175.228,-57.471,-178.108,6.609,148.656
C07135=1179.532,174.979,-57.448,-178.111,6.607,148.656
C07136=1179.537,174.730,-57.426,-178.114,6.606,148.657
C07137=1179.541,174.481,-57.404,-178.116,6.604,148.657
C07138=1179.546,174.232,-57.381,-178.119,6.602,148.657
C07139=1179.551,173.983,-57.359,-178.122,6.600,148.658
C07140=1179.555,173.735,-57.337,-178.124,6.599,148.658
C07141=1179.560,173.485,-57.314,-178.127,6.597,148.659
C07142=1179.564,173.236,-57.292,-178.130,6.595,148.659
C07143=1179.569,172.988,-57.270,-178.132,6.593,148.659
C07144=1179.574,172.738,-57.247,-178.135,6.591,148.660
C07145=1179.579,172.490,-57.226,-178.138,6.590,148.660
C07146=1179.583,172.241,-57.203,-178.140,6.588,148.660
C07147=1179.588,171.991,-57.180,-178.143,6.586,148.661
C07148=1179.593,171.743,-57.158,-178.145,6.584,148.661
C07149=1179.597,171.494,-57.136,-178.148,6.582,148.661
C07150=1179.602,171.245,-57.113,-178.151,6.580,148.662
C07151=1179.606,170.996,-57.091,-178.153,6.579,148.662
C07152=1179.611,170.747,-57.070,-178.157,6.576,148.662
C07153=1179.616,170.498,-57.048,-178.159,6.574,148.663
C07154=1179.621,170.249,-57.025,-178.162,6.573,148.663
C07155=1179.625,170.000,-57.003,-178.165,6.571,148.663
C07156=1179.629,169.751,-56.981,-178.167,6.569,148.664
C07157=1179.634,169.502,-56.959,-178.170,6.567,148.664
C07158=1179.639,169.252,-56.936,-178.173,6.565,148.665
C07159=1179.644,169.004,-56.914,-178.175,6.564,148.665
C07160=1179.648,168.755,-56.892,-178.178,6.562,148.665
C07161=1179.653,168.506,-56.870,-178.181,6.560,148.666
C07162=1179.657,168.257,-56.848,-178.183,6.558,148.666
C07163=1179.663,168.008,-56.826,-178.186,6.557,148.666
C07164=1179.667,167.759,-56.804,-178.189,6.555,148.667
C07165=1179.672,167.510,-56.782,-178.191,6.553,148.667
C07166=1179.676,167.261,-56.760,-178.194,6.551,148.667
C07167=1179.681,167.012,-56.738,-178.197,6.550,148.668
C07168=1179.685,166.763,-56.716,-178.199,6.548,148.668
C07169=1179.690,166.514,-56.695,-178.202,6.546,148.669
C07170=1179.696,166.265,-56.672,-178.205,6.544,148.669
C07171=1179.700,166.016,-56.650,-178.208,6.542,148.669
C07172=1179.705,165.767,-56.629,-178.210,6.541,148.670
C07173=1179.709,165.518,-56.607,-178.213,6.539,148.670
C07174=1179.714,165.269,-56.585,-178.216,6.537,148.670
C07175=1179.718,165.020,-56.563,-178.218,6.535,148.671
C07176=1179.723,164.771,-56.541,-178.221,6.534,148.671
C07177=1179.728,164.522,-56.519,-178.224,6.532,148.672
C07178=1179.732,164.273,-56.497,-178.226,6.530,148.672
C07179=1179.737,164.024,-56.475,-178.229,6.528,148.672
C07180=1179.742,163.775,-56.454,-178.232,6.527,148.673
C07181=1179.746,163.527,-56.432,-178.234,6.525,148.673
C07182=1179.751,163.277,-56.410,-178.237,6.523,148.673
C07183=1179.756,163.028,-56.388,-178.240,6.521,148.674
C07184=1179.761,162.779,-56.366,-178.242,6.519,148.674
C07185=1179.765,162.530,-56.344,-178.245,6.518,148.675
C07186=1179.771,162.281,-56.323,-178.248,6.516,148.675
C07187=1179.775,162.032,-56.301,-178.250,6.514,148.675
C07188=1179.780,161.783,-56.279,-178.253,6.512,148.676
C07189=1179.784,161.534,-56.257,-178.256,6.511,148.676
C07190=1179.788,161.285,-56.236,-178.259,6.509,148.676
C07191=1179.793,161.037,-56.214,-178.261,6.507,148.677
C07192=1179.798,160.787,-56.193,-178.264,6.505,148.677
C07193=1179.802,160.538,-56.171,-178.266,6.504,148.678
C07194=1179.807,160.290,-56.150,-178.269,6.503,148.678
C07195=1179.812,160.040,-56.128,-178.271,6.501,148.678
C07196=1179.817,159.791,-56.107,-178.274,6.499,148.679
C07197=1179.822,159.542,-56.085,-178.277,6.497,148.679
C07198=1179.826,159.293,-56.063,-178.279,6.496,148.679
C07199=1179.831,159.044,-56.041,-178.282,6.494,148.680
C07200=1179.836,158.775,-56.018,-178.285,6.492,148.680
C07201=1179.841,158.506,-55.995,-178.289,6.490,148.681
C07202=1179.846,158.237,-55.972,-178.291,6.488,148.681
C07203=1179.851,157.968,-55.948,-178.294,6.486,148.681
C07204=1179.856,157.719,-55.927,-178.297,6.484,148.682
C07205=1179.861,157.470,-55.906,-178.299,6.483,148.682
C07206=1179.865,157.221,-55.884,-178.302,6.481,148.683
C07207=1179.870,156.972,-55.863,-178.305,6.479,148.683
C07208=1179.875,156.723,-55.842,-178.307,6.477,148.683
C07209=1179.879,156.473,-55.820,-178.310,6.476,148.684
C07210=1179.884,156.225,-55.799,-178.313,6.474,148.684
C07211=1179.889,155.976,-55.777,-178.315,6.473,148.684
C07212=1179.894,155.727,-55.756,-178.318,6.472,148.685
C07213=1179.898,155.478,-55.734,-178.321,6.470,148.685
C07214=1179.903,155.229,-55.713,-178.323,6.468,148.686
C07215=1179.908,154.980,-55.692,-178.326,6.466,148.686
C07216=1179.913,154.731,-55.671,-178.329,6.464,148.687
C07217=1179.917,154.481,-55.649,-178.331,6.463,148.687
C07218=1179.922,154.232,-55.628,-178.334,6.461,148.687
C07219=1179.926,153.984,-55.607,-178.337,6.459,148.688
C07220=1179.932,153.734,-55.586,-178.339,6.457,148.688
C07221=1179.936,153.485,-55.564,-178.342,6.456,148.688
C07222=1179.940,153.236,-55.543,-178.345,6.454,148.689
C07223=1179.945,152.988,-55.522,-178.348,6.452,148.689
C07224=1179.950,152.738,-55.501,-178.350,6.451,148.690
C07225=1179.955,152.489,-55.480,-178.352,6.449,148.690
C07226=1179.959,152.240,-55.458,-178.356,6.448,148.691
C07227=1179.964,151.991,-55.437,-178.358,6.446,148.691
C07228=1179.969,151.742,-55.416,-178.361,6.444,148.691
C07229=1179.973,151.493,-55.395,-178.364,6.443,148.692
C07230=1179.979,151.244,-55.374,-178.366,6.441,148.692
C07231=1179.983,150.995,-55.352,-178.369,6.439,148.692
C07232=1179.987,150.746,-55.332,-178.372,6.437,148.693
C07233=1179.993,150.496,-55.311,-178.374,6.436,148.693
C07234=1179.997,150.248,-55.289,-178.376,6.435,148.694
C07235=1180.002,149.999,-55.269,-178.379,6.433,148.694
C07236=1180.007,149.749,-55.248,-178.382,6.431,148.694
C07237=1180.011,149.500,-55.226,-178.385,6.430,148.695
C07238=1180.016,149.251,-55.205,-178.388,6.428,148.695
C07239=1180.021,149.002,-55.184,-178.390,6.426,148.696
C07240=1180.026,148.753,-55.163,-178.393,6.425,148.696
C07241=1180.030,148.504,-55.142,-178.396,6.423,148.697
C07242=1180.035,148.255,-55.121,-178.398,6.421,148.697
C07243=1180.040,148.006,-55.101,-178.401,6.420,148.697
C07244=1180.044,147.756,-55.080,-178.403,6.418,148.698
C07245=1180.049,147.508,-55.059,-178.406,6.417,148.698
C07246=1180.054,147.259,-55.038,-178.409,6.415,148.699
C07247=1180.059,147.009,-55.017,-178.412,6.413,148.699
C07248=1180.063,146.760,-54.996,-178.415,6.412,148.699
C07249=1180.068,146.511,-54.975,-178.417,6.410,148.700
C07250=1180.073,146.262,-54.955,-178.420,6.408,148.700
C07251=1180.078,146.014,-54.933,-178.422,6.407,148.701
C07252=1180.082,145.765,-54.913,-178.425,6.405,148.701
C07253=1180.087,145.515,-54.892,-178.427,6.404,148.701
C07254=1180.092,145.266,-54.872,-178.431,6.402,148.702
C07255=1180.096,145.016,-54.850,-178.433,6.401,148.702
C07256=1180.101,144.767,-54.830,-178.436,6.399,148.703
C07257=1180.106,144.518,-54.809,-178.439,6.397,148.703
C07258=1180.110,144.269,-54.789,-178.441,6.396,148.703
C07259=1180.116,144.020,-54.768,-178.443,6.394,148.704
C07260=1180.120,143.771,-54.747,-178.446,6.393,148.704
C07261=1180.125,143.522,-54.726,-178.449,6.391,148.705
C07262=1180.129,143.273,-54.705,-178.452,6.389,148.705
C07263=1180.134,143.025,-54.685,-178.455,6.388,148.706
C07264=1180.139,142.775,-54.664,-178.457,6.387,148.706
C07265=1180.143,142.526,-54.643,-178.460,6.385,148.706
C07266=1180.149,142.277,-54.622,-178.462,6.383,148.707
C07267=1180.153,142.027,-54.603,-178.465,6.381,148.707
C07268=1180.159,141.778,-54.582,-178.468,6.380,148.708
C07269=1180.163,141.529,-54.562,-178.471,6.378,148.708
C07270=1180.167,141.280,-54.541,-178.473,6.377,148.709
C07271=1180.173,141.031,-54.520,-178.476,6.376,148.709
C07272=1180.177,140.782,-54.500,-178.478,6.374,148.709
C07273=1180.181,140.533,-54.479,-178.481,6.372,148.710
C07274=1180.187,140.284,-54.458,-178.484,6.371,148.710
C07275=1180.191,140.035,-54.438,-178.487,6.369,148.711
C07276=1180.196,139.786,-54.417,-178.489,6.368,148.711
C07277=1180.201,139.537,-54.397,-178.492,6.366,148.712
C07278=1180.205,139.288,-54.376,-178.494,6.364,148.712
C07279=1180.211,139.038,-54.356,-178.497,6.363,148.712
C07280=1180.215,138.789,-54.336,-178.500,6.361,148.713
C07281=1180.219,138.540,-54.315,-178.503,6.360,148.713
C07282=1180.224,138.291,-54.295,-178.505,6.359,148.714
C07283=1180.229,138.042,-54.274,-178.508,6.357,148.714
C07284=1180.234,137.792,-54.254,-178.510,6.355,148.714
C07285=1180.238,137.543,-54.234,-178.513,6.353,148.715
C07286=1180.243,137.294,-54.213,-178.516,6.352,148.715
C07287=1180.248,137.046,-54.193,-178.518,6.351,148.716
C07288=1180.253,136.796,-54.173,-178.521,6.349,148.716
C07289=1180.258,136.547,-54.153,-178.524,6.348,148.717
C07290=1180.263,136.298,-54.132,-178.527,6.346,148.717
C07291=1180.267,136.049,-54.112,-178.530,6.344,148.718
C07292=1180.272,135.799,-54.092,-178.532,6.343,148.718
C07293=1180.276,135.551,-54.072,-178.535,6.342,148.718
C07294=1180.282,135.301,-54.051,-178.537,6.340,148.719
C07295=1180.286,135.052,-54.031,-178.540,6.338,148.719
C07296=1180.291,134.803,-54.011,-178.543,6.337,148.720
C07297=1180.296,134.555,-53.991,-178.545,6.336,148.720
C07298=1180.301,134.305,-53.971,-178.548,6.334,148.721
C07299=1180.306,134.056,-53.950,-178.551,6.332,148.721
C07300=1180.310,133.807,-53.930,-178.553,6.331,148.721
C07301=1180.315,133.557,-53.910,-178.556,6.330,148.722
C07302=1180.319,133.308,-53.890,-178.559,6.328,148.722
C07303=1180.324,133.059,-53.870,-178.561,6.327,148.723
C07304=1180.329,132.790,-53.848,-178.564,6.325,148.723
